# B&R Automation Studio project mappServicesHighlights
Automation Studio 4.9.3.144 SP; mappServices highlights project; technology packages: mapp 5.12.1, mappView 5.12.1, TextSystem 

## Configuration mappDemoDefault

CPU X20CP1301, AutomationRuntime G4.34, Build 4.1.2, Safety 0.0, Vc V4.72.2

### Task classes (Cpu.sw)
```
Cyclic#1:
  Alarm <- Infrastructure.Alarm.prg [disabled]
  WaterHeate <- WaterHeater.prg [disabled]
  Frequenza <- Frequenza.prg
  Program <- Program.prg
Cyclic#2:
  MainContro <- MainControl.prg [disabled]
  PackML <- Industry.PackML.prg [disabled]
  ConveyorSi <- ConveyorSim.prg [disabled]
Cyclic#6:
  Conteggio <- Conteggio.prg
Cyclic#8:
  Sequence <- Infrastructure.Sequence.prg [disabled]
  IO <- Infrastructure.IO.prg [disabled]
  Report <- Infrastructure.Report.prg
  File <- Infrastructure.File.prg [disabled]  // MpFile sample
  Audit <- Infrastructure.Audit.prg [disabled]  // MpAudit Trail sample
  UserH <- Infrastructure.UserH.prg [disabled]  // MpUser sample
  Recipe <- Infrastructure.Recipe.prg  // MRecipe sample
  Energy <- Infrastructure.Energy.prg [disabled]
  CodeBox <- Infrastructure.CodeBox.prg [disabled]
DataObjects: Arnc0sys
Binaries: TCData, udbdef, arsvcreg, mvLoader, TCLang, arflatprv, arcoal, CfgSeq, OpcUaMap, ashwac, sysconf, CfgEnergy, CfgPackML, CfgHistory, Role, User, CfgRecipe, CfgFile, ashwd, CfgAlarm, iomap, CfgAudit, arconfig, TC, CfgUserXLo, CfgWebXs, asfw, CfgUserX, CfgIO, CfgReportF, CfgReport, CfgCodeCor, CfgComUnit, CfgCodeBox, Config, vcgclass, CfgData, CfgOee, CfgSequenc, vccddbox, vccbtn, vcpdvnc, arialbd, vcmgr, vctcal, vcfile, vcctext, vccnum, Visu02, vcfntttf, vcpkat, vcbclass, vccstr, vclibvc, visvc, vccscale, arial, vccshape, vcalarm, vcpfar00, vcclbox, vcdsloc, vcchtml, Visu01, vccdt, vcchspot, vccbmp, vccpopup, Visu03, vcshared, vcxml, vccurl, vcrt, vccslider, vccgauge, vcctrend, vcnet, vccbar, vccpiech, vcdsint, vcpdsw, vccovl, vccline
Libraries: Runtime, Operator, AsIecCon, astime, AsArSdm, DataObj, FileIO, AsBrStr, AsArLog, sys_lib, brsystem, AsArProf, AsMem, AsWStr, standard, AsBrWStr, ArTextSys, MTTypes, MTBasics, MpAlarmX, MpAudit, MpCom, MpEnergy, MpFile, MpIO, MpPackML, MpRecipe, MpReport, MpSequence, MpUserX, MpWebXs, MpCodeBox, MpServer, MpBase, asstring, aruser, asiomman, ashw, asusb, aseth, arssl, arcert, vcresman, areventlog, arproject, powerlnk
```

### Hardware
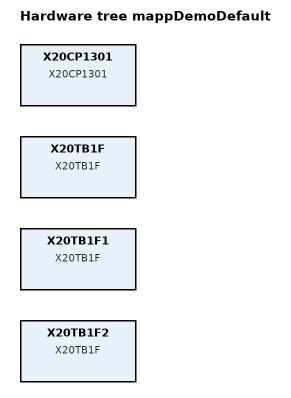
```
X20CP1301 : X20CP1301 v1.7.0.0  [X1 -> X1.SL; X2 -> X2.SL; X3 -> X3.SL]
  Module X1 (Type=X1, Virtual=true, Version=1.7.0.0)
    Connection (Connector=SS1, TargetModule=X20TB1F, TargetConnector=SS)
    Connection (Connector=SL, TargetModule=X20CP1301, TargetConnector=X1)
  Module X2 (Type=X2, Virtual=true, Version=1.7.0.0)
    Connection (Connector=SS1, TargetModule=X20TB1F1, TargetConnector=SS)
    Connection (Connector=SL, TargetModule=X20CP1301, TargetConnector=X2)
  Module X3 (Type=X3, Virtual=true, Version=1.7.0.0)
    Connection (Connector=SS1, TargetModule=X20TB1F2, TargetConnector=SS)
    Connection (Connector=SL, TargetModule=X20CP1301, TargetConnector=X3)
  Connector IF1:
    ActivateIna = 0
  Connector IF2:
    ActivateDevice = 1
    Mode = Manual
    InternetAddress = 192.168.1.38
    SubnetMask = 255.255.255.0
    InaNodeNumber = 0
    Vnc1
    VncKeyMappingFile1 = VC\PS2-Keyboard.dis
    VncMaxConnections1 = 2
    VncRefreshRate1 = 200
  ConfigurationID = mappDemo_CI_Master
  UserPartitionSize = 20
  AutomaticTransferOfUserfiles = on
  RemanentGlobalPvSize = 8192
  VolatileGlobalPvSize = 500000
  CyclicObjects = 300
  BRObjects = 500
  FileDevice1
  FileDeviceName1 = HD
  FileDevicePath1 = C:\
  FileDevice2
  FileDeviceName2 = mappDir
  FileDevicePath2 = C:\mappDemo\CSV
  FileDevice3
  FileDeviceName3 = mappReport
  FileDevicePath3 = C:\mappDemo\Reports\
  FileDevice4
  FileDeviceName4 = mappIO
  FileDevicePath4 = C:\mappDemo\UserFiles\IO
  FileDevice5
  FileDeviceName5 = mappIOBackup
  FileDevicePath5 = C:\mappDemo\UserFiles\IO\Backup
  FileDevice6
  FileDeviceName6 = mappSequence
  FileDevicePath6 = C:\mappDemo\UserFiles\Sequence
  FileDevice7
  FileDeviceName7 = mappCodeBox
  FileDevicePath7 = C:\mappDemo\UserFiles\CodeBox
  FtpUser1
  FtpUsername1 = Promass
  FtpUserPassword1 = NpCmz0K6m8wsjK3Ky3NpfFf+z2PPu3ZJ9pj0GQJGS0g=
  FtpUserSalt1 = EihsEguH
  FTPAccessRight1 = 0
  FTPdevice1 = ALL
  ActivateOpcUa = 1
  OpcUaInformationModels_PV_Version = 1
X20TB1F : X20TB1F v1.0.0.0
X20TB1F1 : X20TB1F v1.0.0.0
X20TB1F2 : X20TB1F v1.0.0.0
```

### IoMap.iom - X20CP1301/IoMap.iom
```iecst
(********************************************************************
 * COPYRIGHT -- Bernecker + Rainer
 ********************************************************************
 * File: IoMap.iom
 * Author: krammerm
 * Created: September 25, 2013
 ********************************************************************
 * IO mapping file
 ********************************************************************)
VAR_CONFIG
	::contatore.Inp_S_Stellare AT %IX."X2".DigitalInput01;
END_VAR
```

### CfgAlarm.mpalarmxcore - X20CP1301/mappServices/CfgAlarm.mpalarmxcore
```
Element gAlarmXCore (Type=mpalarmxcore)
  mapp.AlarmX.Core.Configuration:
    [0]:
      Name = RecordingStarted
      Message = {$mappDemo/MpDataUserAlarm}
      Code = 2501
      Behavior = UserDefined
        AutoReset = TRUE
        Acknowledge = 0
        Recording:
          ActiveToInactive = FALSE
    [1]:
      Name = WaterEmpty
      Message = {$IAT/AlarmWater}
      Code = 2503
      Behavior = LevelMonitoring
        Monitoring:
          MonitoredPV = ::MainContro:Refill.Water
          LowLimitEnable = Static
            Limit = 1
      AdditionalInformation1 = WaterEmpty
    [2]:
      Name = CoffeeEmpty
      Message = {$IAT/AlarmCoffee}
      Code = 2504
      Behavior = LevelMonitoring
        Monitoring:
          MonitoredPV = ::MainContro:Refill.Coffee
          LowLimitEnable = Static
            Limit = 1
      AdditionalInformation1 = CoffeeEmpty
    [3]:
      Name = MilkEmpty
      Message = {$IAT/AlarmMilk}
      Code = 2505
      Behavior = LevelMonitoring
        Monitoring:
          MonitoredPV = ::MainContro:Refill.Milk
          LowLimitEnable = Static
            Limit = 1
      AdditionalInformation1 = MilkEmpty
    [4]:
      Name = SugarEmpty
      Message = {$IAT/AlarmSugar}
      Code = 2506
      Behavior = LevelMonitoring
        Monitoring:
          MonitoredPV = ::MainContro:Refill.Sugar
          LowLimitEnable = Static
            Limit = 1
      AdditionalInformation1 = SugarEmpty
  mapp.AlarmX.Core.Snippets:
    [0]:
      Key = CurrentTemp
      Value:
        PV = ::WaterHeate:WaterHeaterUIConnect.actTemperature
```

### CfgAudit.mpaudittrail - X20CP1301/mappServices/CfgAudit.mpaudittrail
```
Element gAuditTrail (Type=mpaudittrail)
  Audit:
    Events:
      [0] = 16
      [1] = 2
      [2] = 18
      [3] = 17
      [4] = 33
      [5] = 48
      [6] = 64
      [7] = 65
    TextSource = TXT
      OutputFormat = AuditText/Root
      Display = Ne
        Format = AuditDisplayText/DisplayRoot
    Archive = On
    Export:
      FileType = 2
      Encrypt = FALSE
  Alarms = MpAlarmX
```

### CfgCodeBox.mpcodebox - X20CP1301/mappServices/CfgCodeBox.mpcodebox
```
Element CodeBoxCfg (Type=mpcodebox)
  gen:
    progLoc = mappCodeBox
  pvselect:
    0 = 1
      acc = 1
  macro:
    act:
      0:
        id = LampRed
        cd:
          0 = $CodeBox:Lamp.Red := #IN;
      1:
        id = LampYellow
        cd:
          0 = $CodeBox:Lamp.Yellow := #IN;
      2:
        id = LampGreen
        cd:
          0 = $CodeBox:Lamp.Green := #IN;
    cond:
      0:
        id = StartPos
        cd:
          0 = #R := $CodeBox:Cup.StartPosition$;
      1:
        id = CoffeePos
        cd:
          0 = #R := $CodeBox:Cup.CoffeePosition$;
      2:
        id = EndPos
        cd:
          0 = #R := $CodeBox:Cup.EndPosition$;
```

### CfgCodeCor.mpcodeboxcore - X20CP1301/mappServices/CfgCodeCor.mpcodeboxcore
```
Element gCodeBoxCore (Type=mpcodeboxcore)
```

### CfgComUnit.mpcomunit - X20CP1301/mappServices/CfgComUnit.mpcomunit
```
Element gGroup (Type=mpcomunit)
  Display:
    Datapoints:
      0:
        Id = ::Recipe:CoffeeIngredients.Milk
        DisplayUnits:
          Metric:
            Code = MLT
          Imperial:
            Code = MLT
          ImperialUS:
            Code = MLT
      1:
        Id = ::Recipe:CoffeeIngredients.Water
        DisplayUnits:
          Metric:
            Code = MLT
          Imperial:
            Code = MLT
          ImperialUS:
            Code = MLT
      2:
        Id = ::Recipe:CoffeeIngredients.Sugar
        DisplayUnits:
          Metric:
            Code = GRM
          Imperial:
            Code = ONZ
          ImperialUS:
            Code = ONZ
      3:
        Id = ::Recipe:CoffeeIngredients.Coffee
        DisplayUnits:
          Metric:
            Code = GRM
          Imperial:
            Code = ONZ
          ImperialUS:
            Code = ONZ
      4:
        Id = ::Recipe:_Coffee
        DisplayUnits:
          Metric:
            Code = GRM
          Imperial:
            Code = ONZ
          ImperialUS:
            Code = ONZ
      5:
        Id = ::Recipe:_Milk
        DisplayUnits:
          Metric:
            Code = MLT
          Imperial:
            Code = MLT
          ImperialUS:
            Code = MLT
      6:
        Id = ::Recipe:_Sugar
        DisplayUnits:
          Metric:
            Code = GRM
          Imperial:
            Code = ONZ
          ImperialUS:
            Code = ONZ
      7:
        Id = ::Recipe:_Water
        DisplayUnits:
          Metric:
            Code = MLT
          Imperial:
            Code = MLT
          ImperialUS:
            Code = MLT
```

### CfgEnergy.mpenergycore - X20CP1301/mappServices/CfgEnergy.mpenergycore
```
Element gEnergyCore (Type=mpenergycore)
  mapp.energy.collector:
    RecordMemory = 2
    Export:
      FileType:
        ColumnSeparator = ;
  Alarms = MpAlarmX
```

### CfgFile.mpfilemanagerui - X20CP1301/mappServices/CfgFile.mpfilemanagerui
```
Element gFileManagerUI (Type=mpfilemanagerui)
  Alarms = MpAlarmX
```

### CfgHistory.mpalarmxhistory - X20CP1301/mappServices/CfgHistory.mpalarmxhistory
```
Element gAlarmXHistory (Type=mpalarmxhistory)
  mapp.AlarmX.History:
    Auditing = MpAudit
```

### CfgIO.mpio - X20CP1301/mappServices/CfgIO.mpio
```
Element gIoConfig (Type=mpio)
  Import:
    BackupLoc = mappIOBackup
    TemplateLoc = 
  Alarms = MpAlarmX
```

### CfgPackML.mppackmlcore - X20CP1301/mappServices/CfgPackML.mppackmlcore
```
Element gPackMLCore (Type=mppackmlcore)
  Core:
    StartupActiveMode = 1
    Auditing = MpAudit
  Modes:
    Mode[1]:
      ModeID = 1
      Name = Production
      State[1] = 0
      State[5] = 0
      State[10] = 0
      State[11] = 0
      State[12] = 0
      State[13] = 0
      State[14] = 0
      State[17] = 0
    Mode[2]:
      ModeID = 2
  Alarms = MpAlarmX
```

### CfgRecipe.mprecipexml - X20CP1301/mappServices/CfgRecipe.mprecipexml
```
Element gRecipeXml (Type=mprecipexml)
  mapp.Recipe.Xml:
    Auditing = MpAudit
  Alarms = MpAlarmX
```

### CfgReport.mpreportcore - X20CP1301/mappServices/CfgReport.mpreportcore
```
Element gReport (Type=mpreportcore)
  MpReport:
    Settings:
      ResourceDeviceName = HD
      LanguageDependent:
        [0]:
          Language = de
          Font = 1
        [1]:
          Language = en
          Font = 1
    PageLayouts:
      [0]:
        Name = Default
    Styles:
      Text:
        [0]:
          Name = Default
          Size = 12
        [1]:
          Name = Header
          Style = 1
          Size = 20
          Color = FF9900
        [2]:
          Name = Subheader
          Size = 16
          Color = FF9900
      Table:
        [0]:
          Name = Default
          Padding = 10
      Line:
        [0]:
          Name = Default
          Color = FF9900
      Chart:
        PieChart:
          [0]:
            Name = Default
            BorderWidth = 0
        LineChart:
          [0]
        BarChart:
          [0]
    Tables:
      [0]:
        Name = CoffeeInformation
        TableStyle = Default
        TextStyle = Default
        [0]:
          [0] = TextId
            Source = Ora Inizio
            Width = 50
          [1] = DateTime
            Source = ProcessVariable
              ProcessVariable = ::Conteggio:DT_1
            Width = 50
        [1]:
          [0] = TextId
            Source = Ora Fine
            Width = 50
          [1] = DateTime
            Source = ProcessVariable
              ProcessVariable = ::Conteggio:DT_2
            Width = 50
        [2]:
          [0] = TextId
            Source = Tempo Attività
            Width = 50
          [1] = ValueId
            Value:
              ProcessVariable = ::Conteggio:tempo_attuale
            Width = 50
        [3]:
          [0] = TextId
            Source = Giri parziali
            Width = 50
          [1] = ValueId
            Value:
              ProcessVariable = ::contatore.giri_parziali
              UnitDisplay = 1
            Width = 50
        [4]:
          [0] = TextId
            Source = Giri Totali
            Width = 50
          [1] = ValueId
            Value:
              ProcessVariable = ::contatore.giri_totali
              UnitDisplay = 1
            Width = 50
    Contents:
      [0]:
        Name = Discription
        [0]:
          Text = {$Report/ReportDescription}
          TextStyle = Default
      [1]:
        Name = Table
        [0] = Table
          Table = CoffeeInformation
          HorizontalAlign = 1
      [2]:
        Name = Underline
        [0] = Line
          LineStyle = Default
      [3]:
        Name = Header
        [0]:
          Text = {$Report/ReportHeader}
          HorizontalAlign = 1
          TextStyle = Header
      [4]:
        Name = EmptyLine
        [0] = EmptyLine
      [5]:
        Name = EnergyChart
        [0] = Chart
          Chart = Energy
          Width = 60
    Reports:
      [0]:
        Name = Dosaggio
        PageLayout = Default
        Header = Header
        [0]:
          [0]:
            Content = Underline
        [1]:
          [0]:
            Content = EmptyLine
        [2]:
          Heading:
            Text = {$Report/ReportDescriptionHeader}
            TextStyle = Subheader
          [0]:
            Content = Discription
        [3]:
          [0]:
            Content = EmptyLine
        [4]:
          Heading:
            Text = {$Report/ReportHeaderTable}
            TextStyle = Subheader
          [0]:
            Content = Table
        [5]:
          [0]:
            Content = EmptyLine
        [6]:
          [0]:
            Content = EmptyLine
        [7]:
          [0]:
            Content = EnergyChart
  Alarms = MpAlarmX
```

### CfgReportF.mpfilemanagerui - X20CP1301/mappServices/CfgReportF.mpfilemanagerui
```
Element gReportFileManagerUI (Type=mpfilemanagerui)
  Alarms = MpAlarmX
```

### CfgSeq.mpsequencecore - X20CP1301/mappServices/CfgSeq.mpsequencecore
```
Element gSequenceCore (Type=mpsequencecore)
  Sequence:
    DeviceName = mappSequence
    Commands:
      Command[0]:
        Name = SequenceStart
        Text = Start
        Hierarchy = Movement
        CommandType = Movement
          PVStruct = ::Sequence:CmdSeq.Start
      Command[1]:
        Name = SequenceEnd
        Text = End
        Hierarchy = Movement
        CommandType = Movement
          PVStruct = ::Sequence:CmdSeq.Stop
      Command[2]:
        Name = MacroEnd
        Text = EndMakro
        Hierarchy = Movement
      Command[3]:
        Name = Wait
        Text = Wait
        Hierarchy = Movement
        CommandType = Movement
          PVStruct = ::Sequence:CmdSeq.Wait
      Command[4]:
        Name = MoveAxisLeft
        Text = AxisLeft
        Hierarchy = Movement
        CommandType = Movement
          PVStruct = ::Sequence:CmdSeq.AxisLeft
      Command[5]:
        Name = MoveAxisRight
        Text = AxisRight
        Hierarchy = Movement
        CommandType = Movement
          PVStruct = ::Sequence:CmdSeq.AxisRight
          ParStruct = 
      Command[6]:
        Name = Coffee
        Text = Coffee
        Hierarchy = MovementCoffee
        CommandType = Movement
          PVStruct = ::Sequence:CmdSeq.Coffee
      Command[7]:
        Name = TakeOut
        Text = TakeOut
        Hierarchy = MovementCoffee
        CommandType = Movement
          PVStruct = ::Sequence:CmdSeq.TakeOutCup
  Alarms = MpAlarmX
```

### CfgUserX.mpuserx - X20CP1301/mappServices/CfgUserX.mpuserx
```
Element UserMgmtX (Type=mpuserx)
  Groups:
    DefGroup#1:
      id = Administrators
      level = 100
      admin = TRUE
      rights:
        [0] = ViewOnly
        [1] = StartOnly
    DefGroup#2:
      id = Everyone
      level = 1
  Users:
    DefUser#1:
      id = admin
      name = Admin
      lang = en
    DefUser#2:
      id = Anonymous
```

### CfgUserXLo.mpuserxlogin - X20CP1301/mappServices/CfgUserXLo.mpuserxlogin
```
Element gUserXLogin (Type=mpuserxlogin)
  Alarms = MpAlarmX
```

## Logical view

Binary libraries used (declarations not repeated): Runtime, Operator, AsIecCon, AsTime, AsArSdm, DataObj, FileIO, AsBrStr, AsArLog, sys_lib, brsystem, AsWStr, AsArProf, AsMem, standard, AsBrWStr, ArTextSys, MpServer 5.12.0, MpAlarmX 5.12.1, MpBase, MpCodeBox 5.12.1, MpEnergy 5.12.1, MpPackML 5.12.1, MpUserX 5.12.1, MpFile 5.12.1, MpAudit 5.12.1, MpSequence 5.12.1, MpCom, MpIO 5.12.1, MpRecipe 5.12.1, MpWebXs 5.12.1, MpReport 5.12.1, MTBasics, MTTypes, asstring

### Global.typ - Global data types
```iecst
TYPE
	typ_ricetta : 	STRUCT
		Ora_Inizio : DT;
		Ora_Fine : DT;
		Tempo_Attivita : UDINT;
		Giri_Parziali : UDINT;
		Giri_Totali : UDINT;
	END_STRUCT;
	typ_cont : 	STRUCT
		Inp_S_Stellare : BOOL;
		S_stellare : BOOL;
		giri_parziali : UDINT;
		giri_totali : UDINT;
		giri_instant : UDINT;
		frequenza : UDINT;
		nome_ricetta1 : UDINT;
		nome_ricetta2 : STRING[80];
		nome_ricetta3 : UDINT;
		nome_ricetta : STRING[80];
	END_STRUCT;
	PackMLModes :
		(
		PACKML_MODE_PRODUCTION := 1,
		PACKML_MODE_MAINTENANCE := 2
		);
	ReportCoffeeType : 	STRUCT
		Name : STRING[255];
		Water : INT;
		Sugar : INT;
		Coffee : INT;
		Milk : INT;
	END_STRUCT;
	RefillAlarmType : 	STRUCT
		Water : BOOL;
		Sugar : BOOL;
		Milk : BOOL;
		Coffee : BOOL;
	END_STRUCT;
	RefillType : 	STRUCT
		Water : INT;
		Sugar : INT;
		Milk : INT;
		Coffee : INT;
	END_STRUCT;
	CoffeeMainLogicType : 	STRUCT  (*Main logic structure *)
		AxisCupFeeder : CoffeeAxisLogicType; (*Control structure for axis*)
		AxisTakeout : CoffeeAxisLogicType; (*Control structure for axis*)
		cmdAbort : BOOL; (*HMI control to start the brewing process*)
		cmdStop : BOOL; (*HMI control to start the brewing process*)
		cmdClear : BOOL; (*HMI control to start the brewing process*)
		cmdStart : BOOL; (*HMI control to start the brewing process*)
		TemperatureWithinLimit : BOOL; (*HMI control bit *)
		CreateFirstRecipe : BOOL; (*Enable synchronization when creating the default recipes*)
		visPictureIndex : USINT; (*RecipeIndex when creating the default recipes*)
		cmdTakeout : BOOL;
		Refill : RefillType; (*Structure to control the ingredients*)
		AlarmRefill : RefillAlarmType; (*Structure which is controlling the Refill-Alarms*)
		CoffeeState : CoffeeStateEnum;
		ReportCoffee : ARRAY[0..199]OF ReportCoffeeType;
		PackMLState : STRING[80];
		IdleState : BOOL;
	END_STRUCT;
	CoffeeAxisLogicType : 	STRUCT  (*Sub structure for controlling axis*)
		Active : BOOL; (*Axis component is ready*)
		Power : BOOL; (*Power on command*)
		PowerOn : BOOL; (*Power is on*)
		Home : BOOL; (*Homing command *)
		MoveAdditive : BOOL; (*MoveAdditive command*)
		MoveActive : BOOL; (*Move active*)
		InPosition : BOOL; (*Commanded position reached *)
		Position : LREAL; (*Current position*)
	END_STRUCT;
	CoffeeStateEnum :
		(
		COFFEE_WAIT := 0,
		COFFEE_TAKEWATER := 1,
		COFFEE_TAKECOFFEE := 2,
		COFFEE_TAKECOFFEEMILK := 3,
		COFFEE_RELEASE := 4,
		COFFEE_FINISH := 5
		);
END_TYPE
```

### Global.var - Global variables
```iecst
(*Definitions for main components of the coffee machine*)
VAR
	Ricetta : typ_ricetta := (0);
	MpReportCore_0 : MpReportCore := (0); (*Core variable for MpReport*)
	t_ok : BOOL := FALSE;
	CTU_1 : CTU := (0);
	StartGenerate : BOOL := 0; (*variable for interaction with Visualization*)
	gClearAlarm : BOOL := FALSE; (*Check if Alarm can be cleared*)
	gCoffeeMainLogic : CoffeeMainLogicType; (*Control structure of main logic*)
	gSetLanguage : STRING[80] := ''; (*Set the current language*)
	contatore : typ_cont := (0);
END_VAR
```


### Package Logical/Infrastructure - Infrastructure Components

### Program Logical/Infrastructure/Alarm (IEC) - Alarm handling

#### Main.st
```iecst
PROGRAM _CYCLIC

	//Set FB parameter:
	MpAlarmXCore_0(
		Enable := TRUE,
		MpLink := ADR(gAlarmXCore));

	MpAlarmXListUI_0(
		MpLink := ADR(gAlarmXCore),
		Enable := TRUE,
		UIConnect := ADR(MpAlarmXListUIConnect));

	MpAlarmXHistory_0(
		MpLink := ADR(gAlarmXHistory),
		Enable := TRUE,
		DeviceName := ADR('mappDir'),
		Language := ADR(gSetLanguage));

	//Show Alarm-Button in Visualization
	IF MpAlarmXCore_0.ActiveAlarms <> 0 OR MpAlarmXCore_0.PendingAlarms <> 0 THEN
		AlarmButton := 1;
		gCoffeeMainLogic.cmdAbort := TRUE;
		gCoffeeMainLogic.cmdClear := FALSE;
	ELSE
		AlarmButton := 0;
		gCoffeeMainLogic.cmdClear := TRUE;
		gCoffeeMainLogic.cmdAbort := FALSE;
	END_IF

	IF gCoffeeMainLogic.IdleState AND AlarmButton = 0 THEN
		ChangeStyleAlarmButton := 1;
	ELSE
		ChangeStyleAlarmButton := 0;
	END_IF

	IF MpAlarmXHistory_0.CommandDone = TRUE THEN
		MpAlarmXHistory_0.Export := FALSE;
	END_IF

	//Set Alarm-Video
	IF brsstrcmp(ADR(AlarmVideo), ADR("")) = 0 THEN
		AlarmInfo := FALSE;
	ELSE
		AlarmInfo := TRUE;
	END_IF

	FilterConfiguration;
	SortConfiguration;
	HistoryFilter;
	HistorySort;

END_PROGRAM

PROGRAM _EXIT

	//Disable FBs
	MpAlarmXCore_0(Enable := FALSE);
	MpAlarmXHistory_0(Enable := FALSE);
	MpAlarmXHistoryUI_0(Enable := FALSE);
	MpAlarmXListUI_0(Enable := FALSE);

END_PROGRAM
```

#### Variables.var - Local variables
```iecst
VAR
	MpAlarmXHistory_0 : MpAlarmXHistory; (*MpAlarmXHistory instance*)
	MpAlarmXHistoryUI_0 : MpAlarmXHistoryUI; (*MpAlarmXHistoryUI instance*)
	MpAlarmXListUI_0 : MpAlarmXListUI; (*MpAlarmXList instance*)
	MpAlarmXCore_0 : MpAlarmXCore; (*MpAlarmXCore instance*)
	ChangeStyleAlarmButton : USINT := 0; (*changeStyle of a AlarmFlyout in mappView*)
	AlarmButton : BOOL := FALSE; (*Contol Variable for Button in mapp View*)
	MpAlarmXListUIConnect : MpAlarmXListUIConnectType := (0);
	AlarmVideo : WSTRING[255] := "";
	AlarmInfo : BOOL := 0;
	FilterConfiguration : STRING[1000] := '';
	SortConfiguration : STRING[1000] := '';
	HistoryFilter : STRING[2000] := '';
	HistorySort : STRING[2000] := '';
END_VAR
```

### Program Logical/Infrastructure/Recipe (IEC) - Recipe handling

#### Cyclic.ld - Cyclic code
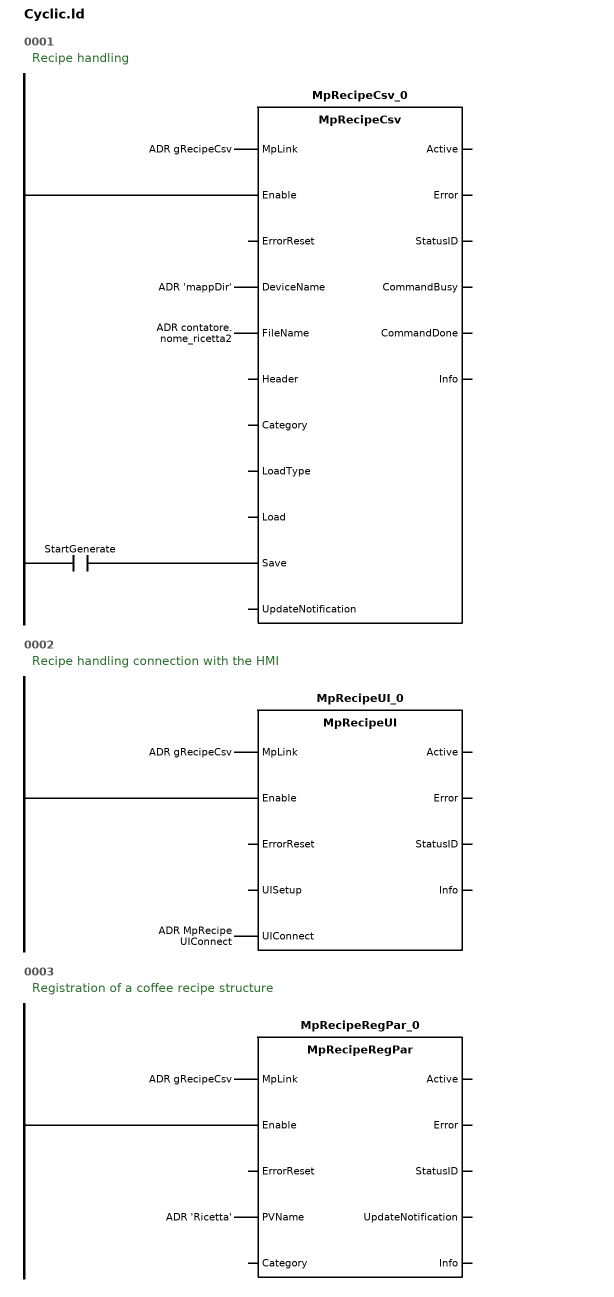
Ladder, written as Structured Text:
```iecst
PROGRAM _CYCLIC
(* Network 1: Recipe handling *)
MpRecipeCsv_0(MpLink := ADR(gRecipeCsv), Enable := TRUE, DeviceName := ADR('mappDir'), FileName := ADR(contatore.nome_ricetta2), Save := StartGenerate);

(* Network 2: Recipe handling connection with the HMI *)
MpRecipeUI_0(MpLink := ADR(gRecipeCsv), Enable := TRUE, UIConnect := ADR(MpRecipeUIConnect));

(* Network 3: Registration of a coffee recipe structure *)
MpRecipeRegPar_0(MpLink := ADR(gRecipeCsv), Enable := TRUE, PVName := ADR('Ricetta'));
END_PROGRAM
```

#### Init.ld - Init code
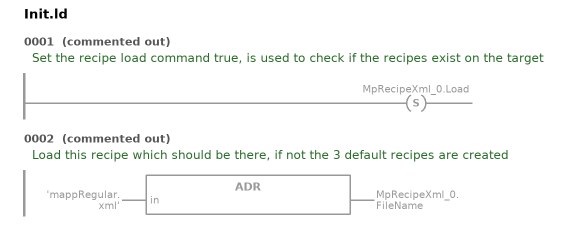
Ladder, written as Structured Text:
```iecst
PROGRAM _INIT
(* Network 1: Set the recipe load command true, is used to check if the recipes exist on the target *) (* commented out *)
// MpRecipeXml_0.Load := TRUE;

(* Network 2: Load this recipe which should be there, if not the 3 default recipes are created *) (* commented out *)
// MpRecipeXml_0.FileName := ADR(in := 'mappRegular.xml');
END_PROGRAM
```

#### Exit.ld
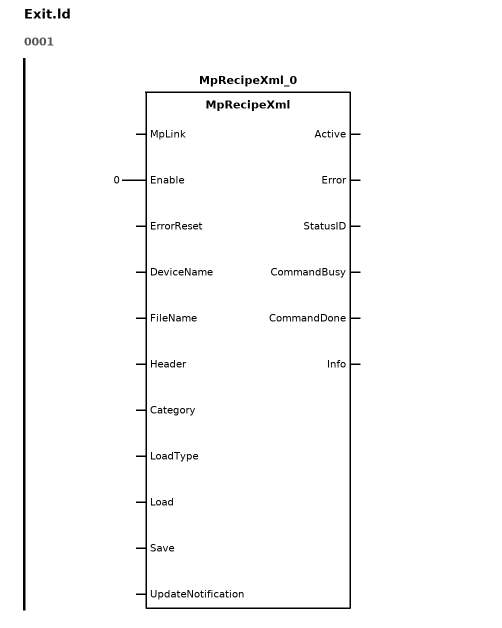
Ladder, written as Structured Text:
```iecst
PROGRAM _EXIT
(* Network 1 *)
MpRecipeXml_0(Enable := 0);
END_PROGRAM
```

#### Variables.var - Local variables
```iecst
VAR
	MpRecipeRegPar_0 : MpRecipeRegPar; (*Registration of the recipe structure variable*)
	MpRecipeUI_0 : MpRecipeUI := (UISetup:=(RecipeListSize:=12,Confirmation:=(RecipeLoad:=0,RecipeSave:=0,RecipeCreate:=0,RecipeDelete:=TRUE))); (*MpRecipeUI Component*)
	MpRecipeCsv_0 : MpRecipeCsv := (0);
	MpRecipeXml_0 : MpRecipeXml; (*Recipe Handling FUB*)
	RecipeCreateStep : RecipeCreateSteps := IDLE; (*Internal variable for recipe creating state machine*)
	MpRecipeUIConnect : MpRecipeUIConnectType := (Recipe:=(Filter:='*xml'),New:=(FileName:='newRecipe.xml')); (*MpRecipeUI connection datapoints*)
	CoffeeIngredients : CoffeeIngredientsType := (Milk:=100,Water:=150,Sugar:=30,Coffee:=60); (*Coffee machine recipe structure*)
END_VAR
(*Variables for AuditTrail*)
VAR
	MpAuditValueChangeStatus : DINT; (*Status variable for MpAuditValueChange function*)
	_Water : INT := 0;
	_Sugar : INT := 0;
	_Milk : INT := 0;
	_Coffee : INT := 0;
	_SelectedIndex : UINT := 800;
END_VAR
```

#### Types.typ - Local Variables
```iecst
TYPE
	RecipeCreateSteps :
		( (*Steps for creating recipes*)
		IDLE := 0, (*Idle State *)
		CREATE_1 := 10, (*Create coffee mappRegular*)
		DONE_1 := 11, (*mappRegular was created*)
		CREATE_2 := 20, (*Create coffee mappEspresso*)
		DONE_2 := 21, (*mappEspresso was created*)
		CREATE_3 := 30, (*Create coffee mappCappuccino*)
		DONE_3 := 31, (*mappCappuccino was created*)
		CREATE_4 := 40, (*Create coffee mappMilkCoffee*)
		DONE_4 := 41, (*mappMilkCoffee was created*)
		ALL_DONE := 50 (*All recipes were created*)
		);
	CoffeeIngredientsType : 	STRUCT  (*Main ingredients structure*)
		Milk : INT; (*Amount of milk per cup*)
		Water : INT; (*Amount of water per cup*)
		Sugar : INT; (*Amount of sugar per cup*)
		Coffee : INT; (*Amount of coffee per cup*)
	END_STRUCT;
END_TYPE
```

#### CreateRecipes.st - Create recipes for the first time the project runs
```iecst
ACTION CreateRecipes:

	// create default recipes in case they don't exist yet on the target
	// recipes are created by using the the MpRecipeXml instance interface

	CASE RecipeCreateStep OF
		IDLE:	// check for load error > triggers the default creation > if no error everything is ready to go
			IF (MpRecipeUIConnect.Recipe.List.Names[0] = '') THEN
				MpRecipeXml_0.Load 			:= FALSE;
				MpRecipeXml_0.ErrorReset 	:= TRUE;
				RecipeCreateStep 			:= CREATE_1;
			ELSE
				MpRecipeUIConnect.Recipe.Load := TRUE;
			END_IF

			// reset the load command from the init when recipe was loaded successfully
			IF (MpRecipeXml_0.CommandDone) AND (MpRecipeXml_0.Load = TRUE) THEN
				MpRecipeXml_0.Load 				:= FALSE;
			END_IF

		CREATE_1:	// create the first recipe with default values, file name and a known picture index (Bitmap Group in the HMI)
			MpRecipeXml_0.ErrorReset 			:= FALSE;

			gCoffeeMainLogic.CreateFirstRecipe 	:= TRUE;
			gCoffeeMainLogic.visPictureIndex	:= 1;
			CoffeeIngredients.Milk 				:= 0;
			CoffeeIngredients.Water 			:= 150;
			CoffeeIngredients.Sugar 			:= 0;
			CoffeeIngredients.Coffee 			:= 60;
			MpRecipeXml_0.FileName 				:= ADR('mappRegular.xml');
			MpRecipeXml_0.Save					:= TRUE;
			RecipeCreateStep 					:= DONE_1;

		DONE_1:	// when CommandDone GoTo next step
			IF(MpRecipeXml_0.CommandDone) THEN
				RecipeCreateStep 			:= CREATE_2;
				MpRecipeXml_0.Save			:= FALSE;
			END_IF;

		CREATE_2:	// create the next recipe with default values, file name and a known picture index (Bitmap Group in the HMI)

			gCoffeeMainLogic.visPictureIndex	:= 2;
			CoffeeIngredients.Milk 				:= 0;
			CoffeeIngredients.Water 			:= 75;
			CoffeeIngredients.Sugar 			:= 0;
			CoffeeIngredients.Coffee 			:= 120;
			MpRecipeXml_0.FileName 				:= ADR('mappEspresso.xml');
			MpRecipeXml_0.Save					:= TRUE;
			RecipeCreateStep 					:= DONE_2;

		DONE_2:	// when CommandDone GoTo next step
			IF (MpRecipeXml_0.CommandDone) THEN
				RecipeCreateStep 			:= CREATE_3;
				MpRecipeXml_0.Save			:= FALSE;
			END_IF;

		CREATE_3:	// create the next recipe with default values, file name and a known picture index (Bitmap Group in the HMI)

			gCoffeeMainLogic.visPictureIndex	:= 3;
			CoffeeIngredients.Milk 				:= 75;
			CoffeeIngredients.Water 			:= 75;
			CoffeeIngredients.Sugar 			:= 20;
			CoffeeIngredients.Coffee 			:= 120;
			MpRecipeXml_0.FileName 				:= ADR('mappCappuccino.xml');
			MpRecipeXml_0.Save					:= TRUE;
			RecipeCreateStep 					:= DONE_3;

		DONE_3:	// when CommandDone creating recipes is done
			IF(MpRecipeXml_0.CommandDone) THEN
				RecipeCreateStep 					:= CREATE_4;
				MpRecipeXml_0.Save					:= FALSE;
			END_IF;
		CREATE_4:	// create the next recipe with default values, file name and a known picture index (Bitmap Group in the HMI)

			gCoffeeMainLogic.visPictureIndex	:= 3;
			CoffeeIngredients.Milk 				:= 100;
			CoffeeIngredients.Water 			:= 50;
			CoffeeIngredients.Sugar 			:= 0;
			CoffeeIngredients.Coffee 			:= 60;
			MpRecipeXml_0.FileName 				:= ADR('mappMilkCoffee.xml');
			MpRecipeXml_0.Save					:= TRUE;
			MpRecipeUIConnect.Recipe.Refresh 	:= TRUE;
			RecipeCreateStep 					:= DONE_4;

		DONE_4:	// when CommandDone creating recipes is done
			IF(MpRecipeXml_0.CommandDone) THEN
				RecipeCreateStep 					:= ALL_DONE;
				MpRecipeXml_0.Save					:= FALSE;
				gCoffeeMainLogic.CreateFirstRecipe 	:= FALSE;
				MpRecipeUIConnect.Recipe.Refresh 	:= FALSE;
			END_IF;
	END_CASE;

END_ACTION
```

#### AuditTrail.st - Watch recipe variable for value change
```iecst
ACTION AuditTrail:

	// Watch for changes in coffee
	IF (CoffeeIngredients.Coffee <> _Coffee) THEN
		MpAuditValueChangeStatus := MpAuditValueChange(gAuditTrail, _Coffee, CoffeeIngredients.Coffee, '100');
		_Coffee 				 := CoffeeIngredients.Coffee;
	END_IF

	// Watch for changes in milk
	IF (CoffeeIngredients.Milk <> _Milk) THEN
		MpAuditValueChangeStatus := MpAuditValueChange(gAuditTrail, _Milk, CoffeeIngredients.Milk, '101');
		_Milk 					 := CoffeeIngredients.Milk;
	END_IF

	// Watch for changes in sugar
	IF (CoffeeIngredients.Sugar <> _Sugar) THEN
		MpAuditValueChangeStatus := MpAuditValueChange(gAuditTrail, _Sugar, CoffeeIngredients.Sugar, '102');
		_Sugar 					 := CoffeeIngredients.Sugar;
	END_IF

	// Watch for changes in water
	IF (CoffeeIngredients.Water <> _Water) THEN
		MpAuditValueChangeStatus := MpAuditValueChange(gAuditTrail, _Water, CoffeeIngredients.Water, '103');
		_Water 					 := CoffeeIngredients.Water;
	END_IF

	//Load new recipe set recipe parameters
	IF MpRecipeUIConnect.Recipe.List.SelectedIndex <> _SelectedIndex THEN
		_SelectedIndex := MpRecipeUIConnect.Recipe.List.SelectedIndex;
		MpRecipeUIConnect.Recipe.Load := TRUE;

	END_IF

	gCoffeeMainLogic.Refill.Coffee := CoffeeIngredients.Coffee ;
	gCoffeeMainLogic.Refill.Milk := CoffeeIngredients.Milk ;
	gCoffeeMainLogic.Refill.Sugar := CoffeeIngredients.Sugar ;
	gCoffeeMainLogic.Refill.Water := CoffeeIngredients.Water ;

END_ACTION
```

### Program Logical/Infrastructure/File (IEC) - File manager

#### Cyclic.ld - Cyclic code
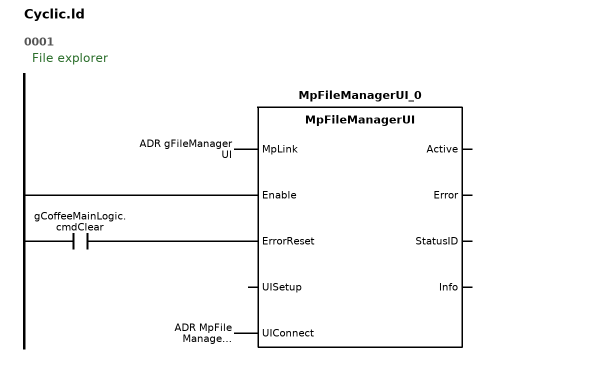
Ladder, written as Structured Text:
```iecst
PROGRAM _CYCLIC
(* Network 1: File explorer *)
MpFileManagerUI_0(MpLink := ADR(gFileManagerUI), Enable := TRUE, ErrorReset := gCoffeeMainLogic.cmdClear, UIConnect := ADR(MpFileManagerUIConnect));
END_PROGRAM
```

#### Init.ld - Init code
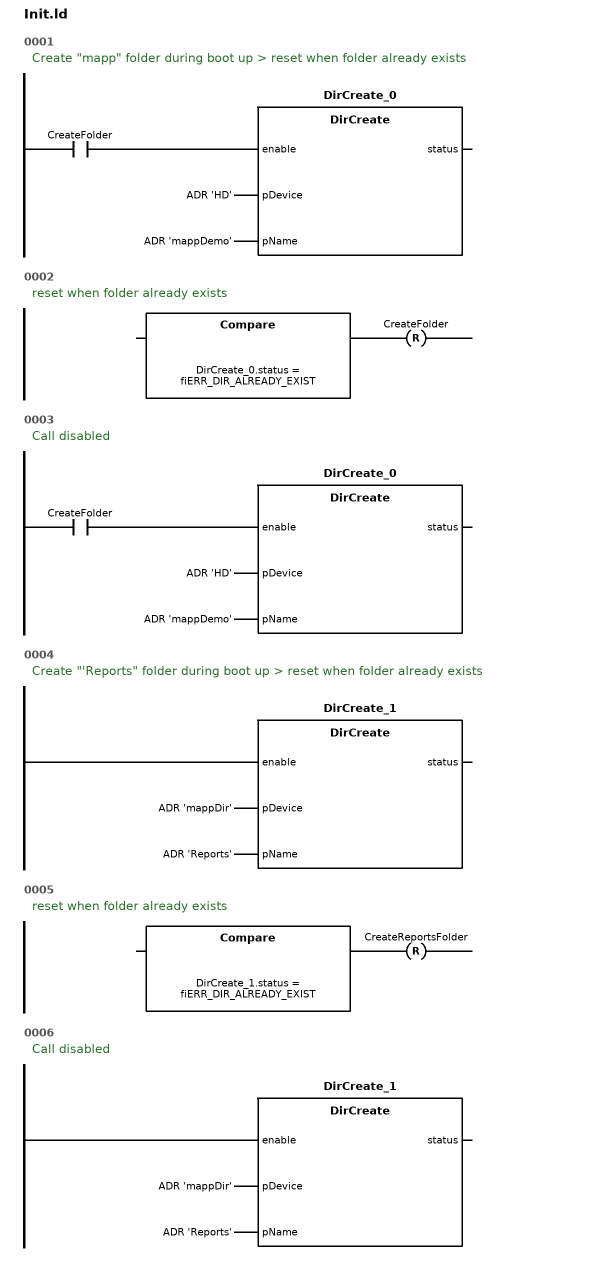
Ladder, written as Structured Text:
```iecst
PROGRAM _INIT
(* Network 1: Create "mapp" folder during boot up > reset when folder already exists  *)
DirCreate_0(enable := CreateFolder, pDevice := ADR('HD'), pName := ADR('mappDemo'));

(* Network 2: reset when folder already exists  *)
IF (DirCreate_0.status = fiERR_DIR_ALREADY_EXIST) THEN CreateFolder := FALSE; END_IF;

(* Network 3: Call disabled *)
DirCreate_0(enable := CreateFolder, pDevice := ADR('HD'), pName := ADR('mappDemo'));

(* Network 4: Create "'Reports" folder during boot up > reset when folder already exists  *)
DirCreate_1(enable := TRUE, pDevice := ADR('mappDir'), pName := ADR('Reports'));

(* Network 5: reset when folder already exists  *)
IF (DirCreate_1.status = fiERR_DIR_ALREADY_EXIST) THEN CreateReportsFolder := FALSE; END_IF;

(* Network 6: Call disabled *)
DirCreate_1(enable := TRUE, pDevice := ADR('mappDir'), pName := ADR('Reports'));
END_PROGRAM
```

#### Variables.var - Local variables
```iecst
VAR
	MpFileManagerUI_0 : MpFileManagerUI; (*MpFileManagerUI instanz*)
	DirCreate_0 : DirCreate; (*FileIO function block for creating the folder "mapp" in case it does not exist yet*)
	CreateFolder : BOOL := TRUE; (*Control bit*)
	MpFileManagerUIConnect : MpFileManagerUIConnectType := (DeviceList:=(DeviceNames:=['mappDir',9('')])); (*MpFileManagerUI connection datapoints*)
	CreateReportsFolder : BOOL := 0;
	DirCreate_1 : DirCreate := (0);
END_VAR
```

### Program Logical/Infrastructure/Audit (IEC) - AuditTrail handling

#### Cyclic.st - Implementation code
```iecst
PROGRAM _CYCLIC

	//Set FB parameters
	MpAuditTrail_0(
		MpLink := ADR(gAuditTrail),
		Enable := TRUE, DeviceName := ADR('mappDir'),
		ErrorReset := gCoffeeMainLogic.cmdClear,
		Language := ADR(gSetLanguage));

	MpAuditTrailUI_0(
		MpLink := ADR(gAuditTrail),
		Enable := TRUE,
		UIConnect := ADR(MpAuditTrailUIConnect),
		ErrorReset := gCoffeeMainLogic.cmdClear,
		Language := ADR(gSetLanguage));

	IF (MpAuditTrail_0.Export) AND (MpAuditTrail_0.CommandDone) THEN
		MpAuditTrail_0.Export := FALSE;
	END_IF

	IF MpAuditTrail_0.ArchiveAvailable THEN
		MpAuditTrail_0.ExportArchive := TRUE;
	ELSE
		MpAuditTrail_0.ExportArchive := FALSE;
	END_IF

	FilterConfiguration;
	SortConfiguraiton;

END_PROGRAM
PROGRAM _EXIT

	//Disable FBs
	MpAuditTrail_0(Enable := FALSE);
	MpAuditTrailUI_0(Enable := FALSE);

END_PROGRAM
```

#### Variables.var - Local variables
```iecst
VAR
	MpAuditTrail_0 : MpAuditTrail; (*Parent component for change tracking*)
	MpAuditTrailUI_0 : MpAuditTrailUI := (UISetup:=(EventListSize:=20)); (*VC4 page connection  *)
	MpAuditTrailUIConnect : MpAuditTrailUIConnectType := (Filter:=(Dialog:=(From:=(Year:=1970,Month:=1,Day:=1,Hour:=00,Minute:=00),Until:=(Year:=1970,Month:=1,Day:=1,Hour:=00,Minute:=00)))); (*MpAuditTrailUI connection datapoints*)
	lng : STRING[80] := '';
	FilterConfiguration : STRING[2000] := '';
	SortConfiguraiton : STRING[2000] := '';
END_VAR
```

### Program Logical/Infrastructure/UserH (IEC) - User handling

#### Main.st
```iecst
PROGRAM _INIT

	LoginAsDefault := FALSE;

END_PROGRAM
PROGRAM _CYCLIC

	//Set FB parameters
	MpUserXLogin_0(
		Enable := TRUE,
		MpLink := ADR(gUserXLogin),
		UserName := ADR(LOGIN_AS_DEFAULT_USERNAME),
		Password := ADR(LOGIN_AS_DEFAULT_PASSWORD));

	MpUserXManagerUI_0(
		Enable := TRUE,
		MpLink := ADR(gUserXLogin),
		UIConnect := ADR(MpUserXManagerUIConnect));

	MpUserXLoginUI_0(
		Enable := TRUE,
		UIConnect := ADR(MpUserXLoginUIConnect),
		MpLink := ADR(gUserXLogin));

	//Call Action
	mappViewConnection;

END_PROGRAM
PROGRAM _EXIT

	//Disable FBs
	MpUserXLogin_0(Enable := FALSE, Login := FALSE);
	MpUserXManagerUI_0(Enable := FALSE);
	MpUserXLoginUI_0(Enable := FALSE);

END_PROGRAM
```

#### mappViewConnection.st - Connection to mapp View
```iecst
ACTION mappViewConnection:

		//Set Login command to FALSE;
	IF MpUserXLogin_0.CommandDone = TRUE THEN
		MpUserXLogin_0.Login := FALSE;
		DeleteTextInput := TRUE ;
	END_IF;

	//Log in as Anonymous
	IF MpUserXLogin_0.CurrentLevel = 0 THEN
		TON_0(IN := TRUE, PT := T#1s5ms);
	ELSIF MpUserXLogin_0.CurrentLevel > 0 THEN
		TON_0(IN := FALSE, PT := T#1s5ms);
	END_IF

	IF ((MpUserXLogin_0.CurrentLevel = 0) AND (LoginAsDefault = TRUE)) OR TON_0.Q = TRUE THEN
		TON_0(IN := FALSE, PT := T#1s5ms);
		MpUserXLogin_0.UserName := ADR(LOGIN_AS_DEFAULT_USERNAME);
		MpUserXLogin_0.Password := ADR(LOGIN_AS_DEFAULT_PASSWORD);
		MpUserXLogin_0.Login := TRUE;
		LoginAsDefault := FALSE;
	END_IF;

	//Set Role in Visualization
	IF MpUserXLogin_0.CurrentLevel = 100 THEN
		Role := 'Administrator';

	ELSIF MpUserXLogin_0.CurrentLevel = 50 THEN
		Role := 'Supervisor';

	ELSIF MpUserXLogin_0.CurrentLevel = 10 THEN
		Role := 'Operator';
	ELSE
		Role := 'Anonymous';
	END_IF

	// Logout in mappView with valuechange in Eventbinding
	IF MpUserXLoginUIConnect.MessageBox.ErrorNumber = 28672 OR MpUserXLoginUIConnect.MessageBox.ErrorNumber = 28673 OR MpUserXLoginUIConnect.MessageBox.ErrorNumber = 28680 THEN
		MappViewLogout := 1;
	ELSIF MpUserXLoginUIConnect.MessageBox.ErrorNumber = 0 THEN
		MappViewLogout := 0;
	END_IF

	IF MpUserXLoginUIConnect.MessageBox.ErrorNumber <> 0 THEN
		ShowErrorLoginDialog := TRUE;
	ELSE
		ShowErrorLoginDialog := FALSE;
	END_IF

END_ACTION
```

#### Variables.var - Local variables
```iecst
VAR CONSTANT
	LOGIN_AS_DEFAULT_USERNAME : WSTRING[20] := "Anonymous"; (*Constant for auto login*)
	LOGIN_AS_DEFAULT_PASSWORD : WSTRING[20] := ""; (*Constant for auto login*)
END_VAR
VAR
	MpUserXManagerUI_0 : MpUserXManagerUI; (*MpUserXManagerUI FUB*)
	MpUserXManagerUIConnect : {REDUND_UNREPLICABLE} MpUserXMgrUIConnectType; (*MpUserXManagerUI connection datapoints*)
	MpUserXLogin_0 : MpUserXLogin := (0); (*MpUserXLogin FUB*)
	MpUserXLoginUI_0 : MpUserXLoginUI := (0); (*MpUserXLoginUI FUB*)
	MpUserXLoginUIConnect : MpUserXLoginUIConnectType := (0); (*MpUserXLoginUI connection datapoints*)
	LoginAsDefault : BOOL := 0; (*trigger login as Anonymous *)
	TON_0 : TON := (0); (*Timer wait for login else login as default*)
	DeleteTextInput : BOOL := 0;
	Role : STRING[80] := '0';
	MappViewLogout : INT := 0;
	ShowErrorLoginDialog : BOOL := 0;
END_VAR
```

### Program Logical/Infrastructure/Energy (IEC) - Energy handling

#### Cyclic.ld - Cyclic code
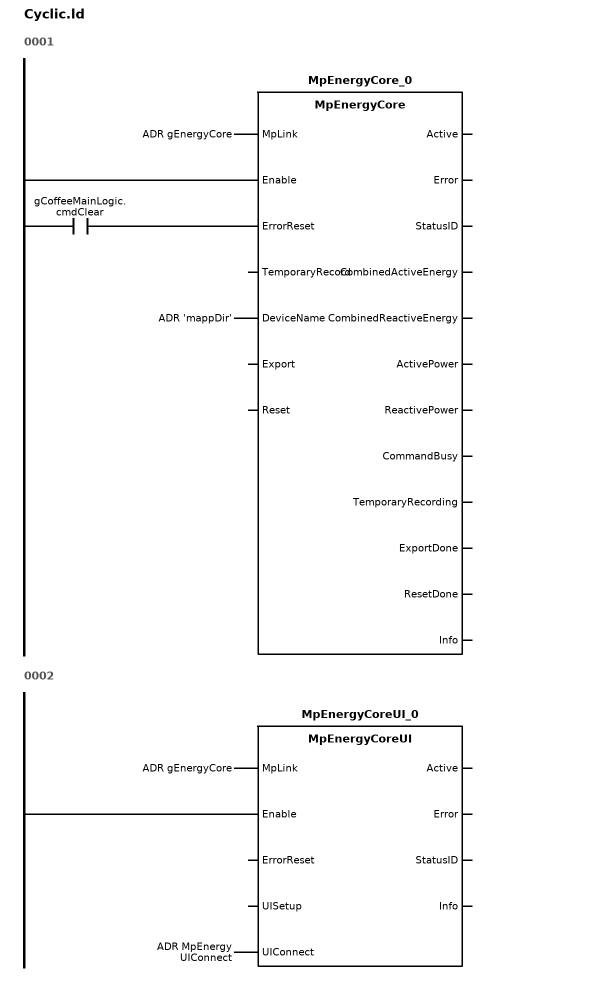
Ladder, written as Structured Text:
```iecst
PROGRAM _CYCLIC
(* Network 1 *)
MpEnergyCore_0(MpLink := ADR(gEnergyCore), Enable := TRUE, ErrorReset := gCoffeeMainLogic.cmdClear, DeviceName := ADR('mappDir'));

(* Network 2 *)
MpEnergyCoreUI_0(MpLink := ADR(gEnergyCore), Enable := TRUE, UIConnect := ADR(MpEnergyUIConnect));
END_PROGRAM
```

#### Exit.ld
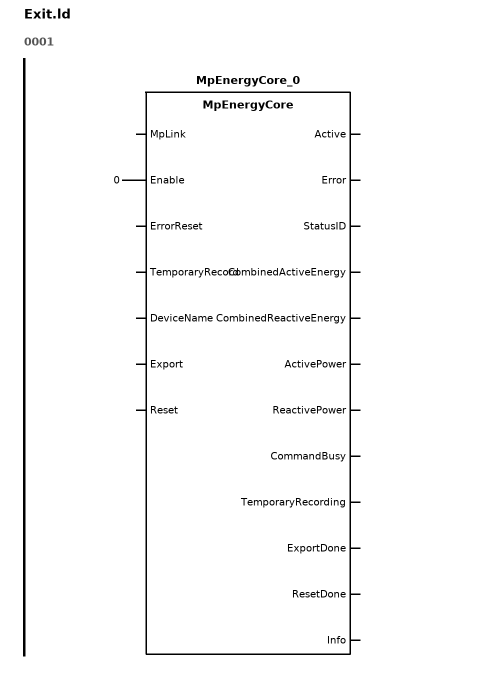
Ladder, written as Structured Text:
```iecst
PROGRAM _EXIT
(* Network 1 *)
MpEnergyCore_0(Enable := 0);
END_PROGRAM
```

#### Variables.var - Local variables
```iecst
VAR
	MpEnergyCore_0 : MpEnergyCore; (*MpEnergyCore instance*)
	MpEnergyCoreUI_0 : MpEnergyCoreUI := (UISetup:=(ModuleListSize:=6)); (*MpEnergyCoreUI instance*)
	MpEnergyUIConnect : MpEnergyCoreUIConnectType; (*MpEnergyUI connection datapoints*)
END_VAR
```

### Program Logical/Infrastructure/Report (IEC) - Report handling

#### Main.st - Cyclic code
```iecst
PROGRAM _CYCLIC

	//Call FBs:
	MpReportCore_0(
		Enable := TRUE,
		MpLink := ADR(gReport),
		Name := ADR(REPORT_NAME),
		DeviceName := ADR(REPORT_DEVICE));
		MpFileManagerUI_0(Enable := TRUE);

	//Call Action
	RefreshReport;

END_PROGRAM
PROGRAM _EXIT

	//Disable FBs
	MpReportCore_0(Enable := FALSE);
	MpFileManagerUI_0(Enable := FALSE);

END_PROGRAM
```

#### Variables.var - Local variables
```iecst
VAR CONSTANT
	STR_FILE_DEVICE : STRING[80] := '/FileDevice:mappReport/';
END_VAR
VAR
	LanguageSelect_0 : LanguageSelect := (LanguageSelection:=['en','de'],SelectedIndex:=0);
	MpFileManagerUI_0 : MpFileManagerUI;
	MpFileManagerUIConnect : MpFileManagerUIConnectType := (DeviceList:=(DeviceNames:=['mappReport',9('')]));
END_VAR
VAR CONSTANT
	REPORT_DEVICE : STRING[80] := 'mappReport'; (*Constant contains filedevice for save reports *)
	REPORT_NAME : STRING[80] := 'Dosaggio'; (*Constant contains name of Report*)
END_VAR
VAR
	DisplayFileName : ARRAY[0..49] OF STRING[255] := [50('')]; (*Displayed Files for mappView*)
	StrSelectedFile : STRING[256] := '0'; (*Gives the path of selected report to pdfViewer in mappView*)
	EnableGenerate : BOOL := TRUE; (*HMI control bit*)
	EnableDelete : BOOL := TRUE; (*HMI control bit*)
	i : USINT := 0; (*index for save filenames in a array*)
	DisplayFileNameIndex : USINT := 0; (*index of selected file for display in table in mappView*)
	DeleteReport : BOOL := 0; (*Start deleting a Report*)
	Refresh : BOOL := 0; (*strrt refresh process*)
	TON_0 : TON := (0); (*Timer to wait before refresh*)
END_VAR
```

#### RefreshReport.st - Showing Report in list
```iecst
ACTION RefreshReport:

	MpFileManagerUI_0.MpLink := ADR(gReportFileManagerUI);
	MpFileManagerUI_0.UIConnect := ADR(MpFileManagerUIConnect);

	IF StartGenerate = TRUE THEN		//Generate process
		MpReportCore_0.Language := ADR(LanguageSelect_0.LanguageSelection[LanguageSelect_0.SelectedIndex]);
		MpReportCore_0.Generate := TRUE;

		IF MpReportCore_0.CommandDone = TRUE THEN

			StartGenerate := FALSE;
			Refresh := TRUE;
			EnableGenerate := FALSE;
		END_IF

	ELSE
		MpReportCore_0.Generate := FALSE;
	END_IF

	IF DeleteReport = TRUE THEN				//Deleting process
		MpFileManagerUIConnect.File.Delete := TRUE;
		MpFileManagerUIConnect.MessageBox.Confirm := TRUE;
		DeleteReport := FALSE;
		Refresh := TRUE;
		EnableDelete := FALSE;
	END_IF

	IF Refresh = TRUE THEN				//Refresh process
		TON_0(IN := TRUE, PT := T#2s);
		IF TON_0.Q = TRUE THEN
			Refresh := FALSE;
			TON_0(IN := FALSE, PT := T#2s);
			MpFileManagerUIConnect.File.Refresh := TRUE;
		END_IF
	END_IF

	IF Refresh = FALSE THEN		//reset enable attribute for buttons
		EnableDelete := TRUE;
		EnableGenerate := TRUE;
	END_IF

	FOR i := 0 TO 49 DO							// Save Filenames to a seperate array for display in Table
		DisplayFileName[i] := MpFileManagerUIConnect.File.List.Items[i].Name;
		IF DisplayFileNameIndex = i THEN		// if selected set a index for display selected file in table
			MpFileManagerUIConnect.File.List.Items[i].IsSelected := TRUE;
		END_IF
	END_FOR

	StrSelectedFile := CONCAT(STR_FILE_DEVICE, MpFileManagerUIConnect.File.List.Items[DisplayFileNameIndex].Name);		// String for pdfViewer to display right report

	IF LanguageSelect_0.SelectedIndex = 0 THEN
		gSetLanguage := 'en';
	ELSE
		gSetLanguage := 'de';
	END_IF

END_ACTION
```

### Program Logical/Infrastructure/IO (IEC) - Hardware handling

#### Main.st - Cyclic code
```iecst
PROGRAM _INIT

	//Enable ImportAllowed
	MpIOImport_0.ImportAllowed := TRUE;

END_PROGRAM
PROGRAM _CYCLIC

	FileName := MpIOImportUIConnect.FileList.Names[MpIOImportUIConnect.FileList.Scroll.SelectedIndex];
	ActiveConfiguration;

	//Set FB parameters
	MpIOImport_0(
		Enable := TRUE,
		MpLink := ADR(gIoConfig),
		DeviceName := ADR('mappIO'),
		FileName := ADR(FileName));

	MpIOImportUI_0(
		Enable := TRUE,
		MpLink := ADR(gIoConfig),
		UIConnect := ADR(MpIOImportUIConnect));

	//Reset Import command if import succeded
	IF MpIOImport_0.CommandDone = TRUE THEN
		MpIOImport_0.Import := FALSE;
	END_IF

END_PROGRAM
PROGRAM _EXIT

	//Disable FBs
	MpIOImport_0(Enable := FALSE, ImportAllowed := FALSE);
	MpIOImportUI_0(Enable := FALSE);

END_PROGRAM
```

#### Variables.var - Local variables
```iecst
VAR
	FileName : STRING[80] := ''; (*FileName of HWConfig file*)
	MpIOImportUIConnect : MpIOImportUIConnectType;
	MpIOImportUI_0 : MpIOImportUI;
	MpIOImport_0 : MpIOImport;
	ActiveConfiguration : STRING[80] := 'Configuration 1';
END_VAR
```

### Program Logical/Infrastructure/Sequence (IEC) - Sequencer handling

#### Types.typ
```iecst
TYPE
	TONType : 	STRUCT
		AxisLeft : TON := (PT:=T#3S);
		TakeOutCup : TON := (PT:=T#3S);
		Coffee : TON := (PT:=T#3S);
		AxisRight : TON := (PT:=T#3S);
		Wait : TON := (PT:=T#3S);
		Start : TON := (PT:=T#1S);
		Stop : TON := (PT:=T#1S);
		ExecuteWait : TON := (PT:=T#2S);
		StopButton : TON;
		CoffeeWait : TON;
	END_STRUCT;
	SequencerStateEnum :
		(
		IDLE,
		MOVE_AXIS_LEFT,
		MOVE_AXIS_RIGHT,
		WAIT,
		COFFEE,
		STOP,
		TAKE_OUT,
		START
		);
	SequencerCommandType : 	STRUCT
		AxisLeft : MpSequencerCommandType;
		Stop : MpSequencerCommandType;
		TakeOutCup : MpSequencerCommandType;
		Coffee : MpSequencerCommandType;
		AxisRight : MpSequencerCommandType;
		Wait : MpSequencerCommandType;
		Start : MpSequencerCommandType;
		End : MpSequencerCommandType;
	END_STRUCT;
END_TYPE
```

#### Variables.var
```iecst
VAR
	Transform : STRING[1000] := '0';
	Timer : TONType := (0);
	SequenceStart : BOOL := 0;
	SavePressed : BOOL := FALSE;
	ParametersCore : MpSequenceCoreParType; (*Parameters for Core function block*)
	MpSequenceCore_0 : MpSequenceCore; (*Inizialize SequencCore function block*)
	EditSequence : BOOL := 0;
	CmdSeq : SequencerCommandType := (0); (*commandstructure for movement command Coffee*)
END_VAR
```

#### Main.st
```iecst
PROGRAM _INIT

	//Enable FBs and set parameters
	MpSequenceCore_0.Enable := TRUE;
	MpSequenceCore_0.Import := TRUE;
	MpSequenceCore_0.Mode := mpSEQUENCE_MODE_SINGLE_CYCLE;
	ParametersCore.Sequence := 'CoffeeSequence.xml';

	Timer.AxisLeft.PT := T#03s;
	Timer.AxisRight.PT := T#03s;
	Timer.Coffee.PT := T#03s;
	Timer.ExecuteWait.PT := T#03s;
	Timer.Start.PT := T#500ms;
	Timer.Stop.PT := T#01s;
	Timer.TakeOutCup.PT := T#01s;
	Timer.Wait.PT := T#03s;
	Timer.StopButton.PT := T#02s;
	Timer.CoffeeWait.PT := T#01s;

END_PROGRAM
PROGRAM _CYCLIC

	//Set FB parameters
	MpSequenceCore_0.MpLink := ADR(gSequenceCore);
	MpSequenceCore_0.Parameters := ADR(ParametersCore);

	IF MpSequenceCore_0.ImportDone THEN
		MpSequenceCore_0.Import := FALSE;
	END_IF

	//Start if Start-Button is pressed
	IF SequenceStart AND MpSequenceCore_0.Info.ReadyToStart THEN
		MpSequenceCore_0.Start := TRUE;
		EditSequence := FALSE;
		MpSequenceCore_0.ErrorReset := FALSE;
	ELSE

		MpSequenceCore_0.Start := FALSE;
		CmdSeq.Start.MovementState := mpSEQUENCE_MOVEMENT_IDLE;
		CmdSeq.AxisLeft.MovementState := mpSEQUENCE_MOVEMENT_IDLE;
		CmdSeq.AxisRight.MovementState := mpSEQUENCE_MOVEMENT_IDLE;
		CmdSeq.Coffee.MovementState := mpSEQUENCE_MOVEMENT_IDLE;
		CmdSeq.End.MovementState := mpSEQUENCE_MOVEMENT_IDLE;
		CmdSeq.TakeOutCup.MovementState := mpSEQUENCE_MOVEMENT_IDLE;
		CmdSeq.Wait.MovementState := mpSEQUENCE_MOVEMENT_IDLE;
		Timer.AxisLeft.IN := FALSE;
		Timer.AxisRight.IN := FALSE;
		Timer.Coffee.IN := FALSE;
		Timer.ExecuteWait.IN := FALSE;
		Timer.Start.IN := FALSE;
		Timer.Stop.IN := FALSE;
		Timer.TakeOutCup.IN := FALSE;
		Timer.Wait.IN := FALSE;
		Timer.StopButton.IN := TRUE;

		Transform := '[{"select":"#g83","duration":1000,"translate":[3.497,-208.81101],"display":true}
		,{"select":"#rect999-9-2","duration":1000,"display":false}
		,{"select":"#rect999-1","duration":1000,"display":false}
		,{"select":"#path49","duration":2000,"fill":7}
		,{"select":"#path39","duration":2000,"fill":0}
		,{"select":"#path41","duration":2000,"fill":2}
		,{"select":"#path3","duration":2000,"fill":3}
		,{"select":"#gLamp1","duration":2000,"fill":7}
		,{"select":"#gLamp2","duration":2000,"fill":7}
		,{"select":"#gLamp3","duration":2000,"fill":7}
		,{"select":"#gLamp4","duration":2000,"fill":7}
		,{"select":"#gLamp5","duration":2000,"fill":7}
		,{"select":"#gLamp6","duration":2000,"fill":7}]';

		IF Timer.StopButton.Q THEN
			Timer.StopButton.IN := FALSE;
		END_IF

		EditSequence := TRUE;

	END_IF

	(****************************************************************START*********************************************************************)
	IF CmdSeq.Start.Start THEN

		CmdSeq.Start.MovementState := mpSEQUENCE_MOVEMENT_ACTIVE;
		Timer.Start.IN := TRUE;
		Transform := '[{"select":"#g83","duration":500,"display":true}]';
		IF Timer.Start.Q THEN
			Timer.Start.IN := FALSE;
			CmdSeq.Start.MovementState := mpSEQUENCE_MOVEMENT_DONE;
		END_IF

	ELSE
		CmdSeq.Start.MovementState := mpSEQUENCE_MOVEMENT_IDLE;
	END_IF

	(****************************************************************AXIS LEFT*********************************************************************)
	IF CmdSeq.AxisLeft.Start THEN

		CmdSeq.AxisLeft.MovementState := mpSEQUENCE_MOVEMENT_ACTIVE;
		Timer.AxisLeft.IN := TRUE;
		Transform := '[{"select":"#g83","duration":3000,"translate":[440,-208.81101]},{"select":"#gLamp1","duration":2000,"fill":8},{"select":"#gLamp4","duration":2000,"fill":8}]';
		IF Timer.AxisLeft.Q THEN
			Timer.AxisLeft.IN := FALSE;
			CmdSeq.AxisLeft.MovementState := mpSEQUENCE_MOVEMENT_DONE;
		END_IF
	ELSE
		CmdSeq.AxisLeft.MovementState := mpSEQUENCE_MOVEMENT_IDLE;
	END_IF

	(****************************************************************AXIS RIGHT*********************************************************************)
	IF CmdSeq.AxisRight.Start THEN

		CmdSeq.AxisRight.MovementState := mpSEQUENCE_MOVEMENT_ACTIVE;
		Timer.AxisRight.IN := TRUE;
		Transform := '[{"select":"#g83","duration":3000,"translate":[560,-208.81101]},{"select":"#gLamp3","duration":2000,"fill":10},{"select":"#gLamp6","duration":2000,"fill":10}]';
		IF Timer.AxisRight.Q THEN
			Timer.AxisRight.IN := FALSE;
			CmdSeq.AxisRight.MovementState := mpSEQUENCE_MOVEMENT_DONE;
		END_IF
	ELSE
		CmdSeq.AxisRight.MovementState := mpSEQUENCE_MOVEMENT_IDLE;
	END_IF

	(****************************************************************COFFEE*********************************************************************)
	IF CmdSeq.Coffee.Start THEN

		CmdSeq.Coffee.MovementState := mpSEQUENCE_MOVEMENT_ACTIVE;
		Timer.Coffee.IN := TRUE;
		Transform :='[{"select":"#path39","duration":2000,"fill":7}
		,{"select":"#path41","duration":2000,"fill":7}
		,{"select":"#path3","duration":2000,"fill":7}
		,{"select":"#gLamp2","duration":2000,"fill":9},
		{"select":"#gLamp5","duration":2000,"fill":9}]';
		IF Timer.Coffee.Q THEN

			Timer.ExecuteWait.IN := TRUE;

			Transform := '[{"select":"#rect999-9-2","duration":2000,"display":true,"fill":1}
			,{"select":"#rect999-1","duration":2000,"display":true,"fill":1}
			,{"select":"#path49","duration":2000,"fill":0}
			,{"select":"#path39","duration":2000,"fill":0}
			,{"select":"#path41","duration":2000,"fill":2}
			,{"select":"#path3","duration":2000,"fill":3}]';
			IF Timer.ExecuteWait.Q THEN

				Timer.CoffeeWait.IN := TRUE;
				Transform := '[{"select":"#rect999-1","duration":1000,"display":false},
				{"select":"#rect999-9-2","duration":1000,"display":false},
				{"select":"#path49","duration":1000,"fill":7}]';
				IF Timer.CoffeeWait.Q THEN
					Timer.CoffeeWait.IN := FALSE;
					Timer.Coffee.IN := FALSE;
					Timer.ExecuteWait.IN := FALSE;
					CmdSeq.Coffee.MovementState := mpSEQUENCE_MOVEMENT_DONE;
				END_IF
			END_IF
		END_IF

	ELSE
		CmdSeq.Coffee.MovementState := mpSEQUENCE_MOVEMENT_IDLE;
	END_IF

	(****************************************************************TAKEOUT*********************************************************************)
	IF CmdSeq.TakeOutCup.Start THEN

		CmdSeq.TakeOutCup.MovementState := mpSEQUENCE_MOVEMENT_ACTIVE;
		Timer.TakeOutCup.IN := TRUE;
		Transform := '[{"select":"#g83","duration":500,"display":false}]';
		IF Timer.TakeOutCup.Q THEN
			Timer.TakeOutCup.IN := FALSE;
			CmdSeq.TakeOutCup.MovementState := mpSEQUENCE_MOVEMENT_DONE;
		END_IF
	ELSE
		CmdSeq.TakeOutCup.MovementState := mpSEQUENCE_MOVEMENT_IDLE;
	END_IF

	(****************************************************************WAIT*********************************************************************)
	IF CmdSeq.Wait.Start THEN
		CmdSeq.Wait.MovementState := mpSEQUENCE_MOVEMENT_ACTIVE;
		Timer.Wait.IN := TRUE;

		IF Timer.Wait.Q THEN
			Timer.Wait.IN := FALSE;
			CmdSeq.Wait.MovementState := mpSEQUENCE_MOVEMENT_DONE;
		END_IF
	ELSE
		CmdSeq.Wait.MovementState := mpSEQUENCE_MOVEMENT_IDLE;
	END_IF

	(****************************************************************STOP*********************************************************************)
	IF CmdSeq.Stop.Start THEN
		CmdSeq.Stop.MovementState := mpSEQUENCE_MOVEMENT_ACTIVE;
		Timer.Stop.IN := TRUE;
		Transform := '[{"select":"#g83","duration":1000,"translate":[3.497,-208.81101]}
		]';

		IF Timer.Stop.Q THEN
			Timer.Stop.IN := FALSE;
			CmdSeq.Stop.MovementState := mpSEQUENCE_MOVEMENT_DONE;
			Transform := '[{"select":"#g83","duration":500,"display":true}]';
			SequenceStart := FALSE;
		END_IF
	ELSE
		CmdSeq.Stop.MovementState := mpSEQUENCE_MOVEMENT_IDLE;
	END_IF

	(****************************************************************ERROR*********************************************************************)
	IF MpSequenceCore_0.Error THEN
		SequenceStart := FALSE;
		MpSequenceCore_0.Import := FALSE;
		MpSequenceCore_0.ErrorReset := gCoffeeMainLogic.cmdClear;
	END_IF

	IF SavePressed THEN
		MpSequenceCore_0.Import := TRUE;
		SavePressed := FALSE;
	END_IF

	//Call FB
	MpSequenceCore_0();
	Timer.AxisLeft();
	Timer.AxisRight();
	Timer.Coffee();
	Timer.Start();
	Timer.Stop();
	Timer.TakeOutCup();
	Timer.Wait();
	Timer.ExecuteWait();
	Timer.StopButton();
	Timer.CoffeeWait();

END_PROGRAM
PROGRAM _EXIT

	//Disable FB
	MpSequenceCore_0(Enable := FALSE);

END_PROGRAM
```

### Program Logical/Infrastructure/CodeBox (IEC) - CodeBox handling

#### Main.st - Init, cyclic, exit code
```iecst
PROGRAM _INIT

	State := WAIT;

END_PROGRAM

PROGRAM _CYCLIC

	//Set FB parameter
	MpCodeBoxCore_0(
	MpLink := ADR(gCodeBoxCore),
	Enable := TRUE,
	ErrorReset := gCoffeeMainLogic.cmdClear);

	Cup;
	Lamp;

	CodeBoxTransform;

	CASE State OF
		WAIT:
			CodeBoxTransform := '[{"select":"#gLamp1","duration":200,"fill":7}
			,{"select":"#gLamp2","duration":200,"fill":7}
			,{"select":"#gLamp3","duration":200,"fill":7}
			,{"select":"#gLamp4","duration":200,"fill":7}
			,{"select":"#gLamp5","duration":200,"fill":7}
			,{"select":"#gLamp6","duration":200,"fill":7}]';

			IF gCoffeeMainLogic.PackMLState = 'Idle' THEN
				State := CUP_START_POS;

			END_IF

		CUP_START_POS:
			Cup.StartPosition := TRUE;
			IF Lamp.Green THEN

				CodeBoxTransform := '[{"select":"#gLamp1","duration":1000,"fill":10}
					,{"select":"#gLamp2","duration":1000,"fill":7}
					,{"select":"#gLamp3","duration":1000,"fill":7}
					,{"select":"#gLamp4","duration":1000,"fill":10}
					,{"select":"#gLamp5","duration":1000,"fill":7}
					,{"select":"#gLamp6","duration":1000,"fill":7}]';

			ELSIF Lamp.Red THEN
				CodeBoxTransform := '[{"select":"#gLamp1","duration":1000,"fill":8}
				,{"select":"#gLamp2","duration":1000,"fill":7}
				,{"select":"#gLamp3","duration":1000,"fill":7}
				,{"select":"#gLamp4","duration":1000,"fill":8}
				,{"select":"#gLamp5","duration":1000,"fill":7}
				,{"select":"#gLamp6","duration":1000,"fill":7}]';

			ELSIF Lamp.Yellow THEN
				CodeBoxTransform := '[{"select":"#gLamp1","duration":1000,"fill":9}
				,{"select":"#gLamp2","duration":1000,"fill":7}
				,{"select":"#gLamp3","duration":1000,"fill":7}
				,{"select":"#gLamp4","duration":1000,"fill":9}
				,{"select":"#gLamp5","duration":1000,"fill":7}
				,{"select":"#gLamp6","duration":1000,"fill":7}]';
			ELSE
				CodeBoxTransform := '[{"select":"#gLamp1","duration":1000,"fill":7}
				,{"select":"#gLamp2","duration":1000,"fill":7}
				,{"select":"#gLamp3","duration":1000,"fill":7}
				,{"select":"#gLamp4","duration":1000,"fill":7}
				,{"select":"#gLamp5","duration":1000,"fill":7}
				,{"select":"#gLamp6","duration":1000,"fill":7}]';
			END_IF

			IF gCoffeeMainLogic.PackMLState = 'Execute' THEN
				State := CUP_COFFEE;
				Cup.StartPosition := FALSE;
			END_IF

		CUP_COFFEE:
			Cup.CoffeePosition := TRUE;
			IF gCoffeeMainLogic.PackMLState = 'Completing' THEN
				State := CUP_END_POS;
				Cup.CoffeePosition := FALSE;
			END_IF

			IF Lamp.Green THEN

				CodeBoxTransform := '[{"select":"#gLamp1","duration":1000,"fill":7}
				,{"select":"#gLamp2","duration":1000,"fill":10}
				,{"select":"#gLamp3","duration":1000,"fill":7}
				,{"select":"#gLamp4","duration":1000,"fill":7}
				,{"select":"#gLamp5","duration":1000,"fill":10}
				,{"select":"#gLamp6","duration":1000,"fill":7}]';

			ELSIF Lamp.Red THEN
				CodeBoxTransform := '[{"select":"#gLamp1","duration":1000,"fill":7}
				,{"select":"#gLamp2","duration":1000,"fill":8}
				,{"select":"#gLamp3","duration":1000,"fill":7}
				,{"select":"#gLamp4","duration":1000,"fill":7}
				,{"select":"#gLamp5","duration":1000,"fill":8}
				,{"select":"#gLamp6","duration":1000,"fill":7}]';

			ELSIF Lamp.Yellow THEN
				CodeBoxTransform := '[{"select":"#gLamp1","duration":1000,"fill":7}
				,{"select":"#gLamp2","duration":1000,"fill":9}
				,{"select":"#gLamp3","duration":1000,"fill":7}
				,{"select":"#gLamp4","duration":1000,"fill":7}
				,{"select":"#gLamp5","duration":1000,"fill":9}
				,{"select":"#gLamp6","duration":1000,"fill":7}]';
			ELSE
				CodeBoxTransform := '[{"select":"#gLamp1","duration":1000,"fill":7}
				,{"select":"#gLamp2","duration":1000,"fill":7}
				,{"select":"#gLamp3","duration":1000,"fill":7}
				,{"select":"#gLamp4","duration":1000,"fill":7}
				,{"select":"#gLamp5","duration":1000,"fill":7}
				,{"select":"#gLamp6","duration":1000,"fill":7}]';
			END_IF
		CUP_END_POS:
			Cup.EndPosition := TRUE;
			IF Lamp.Green THEN

				CodeBoxTransform := '[{"select":"#gLamp1","duration":1000,"fill":7}
				,{"select":"#gLamp2","duration":1000,"fill":7}
				,{"select":"#gLamp3","duration":1000,"fill":10}
				,{"select":"#gLamp4","duration":1000,"fill":7}
				,{"select":"#gLamp5","duration":1000,"fill":7}
				,{"select":"#gLamp6","duration":1000,"fill":10}]';

			ELSIF Lamp.Red THEN
				CodeBoxTransform := '[{"select":"#gLamp1","duration":1000,"fill":7}
				,{"select":"#gLamp2","duration":1000,"fill":7}
				,{"select":"#gLamp3","duration":1000,"fill":8}
				,{"select":"#gLamp4","duration":1000,"fill":7}
				,{"select":"#gLamp5","duration":1000,"fill":7}
				,{"select":"#gLamp6","duration":1000,"fill":8}]';

			ELSIF Lamp.Yellow THEN
				CodeBoxTransform := '[{"select":"#gLamp1","duration":1000,"fill":7}
				,{"select":"#gLamp2","duration":1000,"fill":7}
				,{"select":"#gLamp3","duration":1000,"fill":9}
				,{"select":"#gLamp4","duration":1000,"fill":7}
				,{"select":"#gLamp5","duration":1000,"fill":7}
				,{"select":"#gLamp6","duration":1000,"fill":9}]';
			ELSE
				CodeBoxTransform := '[{"select":"#gLamp1","duration":1000,"fill":7}
				,{"select":"#gLamp2","duration":1000,"fill":7}
				,{"select":"#gLamp3","duration":1000,"fill":7}
				,{"select":"#gLamp4","duration":1000,"fill":7}
				,{"select":"#gLamp5","duration":1000,"fill":7}
				,{"select":"#gLamp6","duration":1000,"fill":7}]';
			END_IF
			IF gCoffeeMainLogic.PackMLState = 'Idle' THEN
				State := WAIT;
				Cup.EndPosition := FALSE;
			END_IF

	END_CASE

END_PROGRAM

PROGRAM _EXIT

	MpCodeBoxCore_0(Enable := FALSE);

END_PROGRAM
```

#### Types.typ - Local data types
```iecst
TYPE
	CodeBox_State :
		(
		WAIT := 0,
		CUP_COFFEE := 1,
		CUP_END_POS := 2,
		CUP_START_POS := 3
		);
	Cup_Type : 	STRUCT
		StartPosition : BOOL;
		EndPosition : BOOL;
		CoffeePosition : BOOL;
	END_STRUCT;
	Lamp_type : 	STRUCT
		Red : BOOL;
		Yellow : BOOL;
		Green : BOOL;
	END_STRUCT;
END_TYPE
```

#### Variables.var - Local variables
```iecst
VAR
	State : CodeBox_State := CUP_START_POS;
	Cup : Cup_Type := (0);
	MpCodeBoxCore_0 : MpCodeBoxCore := (0);
	Lamp : Lamp_type := (0);
	CodeBoxTransform : STRING[2000] := '';
END_VAR
```

- Project.language (not shown)

### Package Logical/Industry - Industry Components

### Program Logical/Industry/PackML (IEC) - PackML handling

#### Variables.var
```iecst
VAR
	MpPackMLBasicUI_0 : MpPackMLBasicUI; (*MpPackMLBasicUI instance*)
	MpPackMLBasicUIConnect : MpPackMLBasicUIConnectType := (ModeControl:=(SelectedIndex:=1)); (*MpPackMLBasicUI UI connection datapoints*)
	MpPackMLStatisticsUI_0 : MpPackMLStatisticsUI; (*MpPackMLStatisticsUI instance*)
	MpPackMLStatisticsUIConnect : MpPackMLStatisticsUIConnectType; (*MpPackMLStatistics UI connection datapoints*)
	MpPackMLMode_0 : MpPackMLMode;
	MpPackMLCore_0 : MpPackMLCore;
	MpPackMLMode_1 : MpPackMLMode;
END_VAR
```

#### Main.st
```iecst
PROGRAM _CYCLIC

	//Set FB parameters
	MpPackMLCore_0(
		MpLink := ADR(gPackMLCore),
		Enable := TRUE);

	MpPackMLMode_0(
		MpLink := ADR(gPackMLCore),
		Enable := TRUE,
		ModeID := PACKML_MODE_PRODUCTION,
		Start := gCoffeeMainLogic.cmdStart,
		Stop := gCoffeeMainLogic.cmdStop,
		Reset := MpPackMLStateIsActive(gPackMLCore,mpPACKML_STATE_STOPPED,PACKML_MODE_PRODUCTION),
		Abort := (gCoffeeMainLogic.cmdAbort AND MpPackMLMode_0.ModeActive),
		Clear := gCoffeeMainLogic.cmdClear);

	MpPackMLMode_1(
		MpLink := ADR(gPackMLCore),
		Enable := TRUE,
		ModeID := PACKML_MODE_MAINTENANCE);

	MpPackMLBasicUI_0(
		MpLink := ADR(gPackMLCore),
		Enable := TRUE,
		UIConnect := ADR(MpPackMLBasicUIConnect));

	MpPackMLStatisticsUI_0(
		MpLink := ADR(gPackMLCore),
		Enable := TRUE,
		UIConnect := ADR(MpPackMLStatisticsUIConnect));

	//Check if you can refill the ingredients
	IF MpPackMLCore_0.Info.StateCurrent = 'Idle' OR MpPackMLCore_0.Info.StateCurrent = 'Aborted' THEN
		gCoffeeMainLogic.IdleState := TRUE;
	ELSE
		gCoffeeMainLogic.IdleState := FALSE;
	END_IF

END_PROGRAM
PROGRAM _EXIT

	//Disable FBs
	MpPackMLCore_0(Enable := FALSE);
	MpPackMLMode_0(Enable := FALSE);
	MpPackMLMode_1(Enable := FALSE);
	MpPackMLBasicUI_0(Enable := FALSE);
	MpPackMLStatisticsUI_0(Enable := FALSE);

END_PROGRAM
```

### Program Logical/MainControl (IEC) - MainContol program

#### Cyclic.st - Cyclic code
```iecst
PROGRAM _CYCLIC

	// Main state machine for the brewing process handled by PackML

(****************************************************************IDLE*********************************************************************)

	IF (MpPackMLStateIsActive(gPackMLCore, mpPACKML_STATE_IDLE, PACKML_MODE_PRODUCTION)) THEN
		gCoffeeMainLogic.PackMLState := 'Idle';
		TransitionTime := 500;
		TransformTime := T#500ms;
		gCoffeeMainLogic.AxisCupFeeder.Power 		:= TRUE;
		gCoffeeMainLogic.AxisTakeout.Power 			:= TRUE;

		IF (gCoffeeMainLogic.AxisTakeout.Active = TRUE) AND (gCoffeeMainLogic.AxisCupFeeder.Active = TRUE)  THEN

			MainCoffeeUIConnect.visShowButtonStart 	:= YES;
			MainCoffeeUIConnect.visWaterLevel 		:= 100;	// initialize water level
			Transform := '[{"select":"#g83","duration":500,"display":true}]';
		ELSE

			gCoffeeMainLogic.cmdAbort := TRUE;

		END_IF

	END_IF

	(****************************************************************RESETTING*********************************************************************)

	IF (MpPackMLStateIsActive(gPackMLCore, mpPACKML_STATE_RESETTING
		, PACKML_MODE_PRODUCTION)) THEN
		gCoffeeMainLogic.PackMLState := 'Resetting';
		gCoffeeMainLogic.cmdClear 		:= FALSE;
		gCoffeeMainLogic.cmdAbort 		:= FALSE;

		gCoffeeMainLogic.AxisCupFeeder.Power 		:= TRUE;				// power and home both conveyor axes
		gCoffeeMainLogic.AxisTakeout.Power 			:= TRUE;

		IF(gCoffeeMainLogic.AxisTakeout.PowerOn = TRUE) AND (gCoffeeMainLogic.AxisCupFeeder.PowerOn = TRUE)  THEN

			MpPackMLStateComplete(gPackMLCore, PACKML_MODE_PRODUCTION);

		END_IF
	END_IF

	(******************************************************************STARTING*******************************************************************)

	IF (MpPackMLStateIsActive(gPackMLCore, mpPACKML_STATE_STARTING, PACKML_MODE_PRODUCTION)) THEN
		gCoffeeMainLogic.PackMLState := 'Starting';
		MainCoffeeUIConnect.visShowMainBrewing 			:= YES;
		MainCoffeeUIConnect.visShowMainRecipe  			:= YES;
		MainCoffeeUIConnect.visShowButtonStart 			:= NO;
		MainCoffeeUIConnect.visCupSlider 				:= 0;

		TransitionTime := 3000;
		Transform := '[{"select":"#g83","duration":3000,"translate":[375,-87.299533]}]';
		TransformTime := T#3S;
		TransformWait.IN := TRUE;
		TransformWait.PT := TransformTime;

		gCoffeeMainLogic.AxisCupFeeder.MoveAdditive 	:= TRUE;			// start moving the cup to fill station
		gCoffeeMainLogic.cmdStart := FALSE;

		IF (gCoffeeMainLogic.AxisCupFeeder.InPosition) AND TransformWait.Q = TRUE THEN
			TransformWait.IN := FALSE;
			gCoffeeMainLogic.AxisCupFeeder.MoveAdditive 	:= FALSE;				// reset command when in position
			MainCoffeeUIConnect.visCupSlider 				:= 1000;
			gCoffeeMainLogic.AxisCupFeeder.InPosition := FALSE;
			gCoffeeMainLogic.AxisCupFeeder.Position 	:= 0.0;
			MpPackMLStateComplete(gPackMLCore, PACKML_MODE_PRODUCTION);
			TransformWait();
		END_IF

	END_IF

	(******************************************************************EXECUTE*******************************************************************)

	IF (MpPackMLStateIsActive(gPackMLCore, mpPACKML_STATE_EXECUTE, PACKML_MODE_PRODUCTION)) THEN
		gCoffeeMainLogic.PackMLState := 'Execute';
		TransitionTime := 3000;
		TransformTime := T#3S;
		Transform :='[{"select":"#path39","duration":2000,"fill":7}
		,{"select":"#path41","duration":2000,"fill":7}
		,{"select":"#path3","duration":2000,"fill":7}
		,{"select":"#rect999","duration":2000,"display":true,"fill":1}
		,{"select":"#rect999-9","duration":2000,"display":true,"fill":1}
		,{"select":"#path49","duration":2000,"fill":0}]';
		ExecuteWait.IN := TRUE;
		ExecuteWait.PT := TransformTime;
		ExecuteWait();

		IF ExecuteWait.Q = TRUE THEN
			FillCoffeeWait.IN := TRUE;
			FillCoffeeWait.PT := T#2s;
			Transform := '[{"select":"#path49","duration":2000,"fill":0}
			,{"select":"#path39","duration":2000,"fill":0}
			,{"select":"#path41","duration":2000,"fill":2}
			,{"select":"#path3","duration":2000,"fill":3}
			,{"select":"#rect999","duration":500,"display":false}
			,{"select":"#rect999-9","duration":500,"display":false}
			,{"select":"#path49","duration":2000,"fill":7}]';

			IF FillCoffeeWait.Q THEN
				FillCoffeeWait.IN := FALSE;
				ExecuteWait.IN := FALSE;
				gCoffeeMainLogic.AxisTakeout.MoveAdditive := TRUE;					// start moving cup to take out
				MpPackMLStateComplete(gPackMLCore, PACKML_MODE_PRODUCTION);
			END_IF
		END_IF

	END_IF

	(******************************************************************Completing*******************************************************************)

	IF (MpPackMLStateIsActive(gPackMLCore, mpPACKML_STATE_COMPLETING, PACKML_MODE_PRODUCTION)) THEN
		TransitionTime := 3000;
		Transform := '[{"select":"#g83","duration":3000,"translate":[560,-87.299533]}]';
		gCoffeeMainLogic.PackMLState := 'Completing';
		TransformWait.IN := TRUE;
		TransformWait.PT := TransformTime;

		IF (gCoffeeMainLogic.AxisTakeout.InPosition) AND TransformWait.Q = TRUE THEN

			TransitionTime := 500;
			Transform := '[{"select":"#g83","duration":500,"display":false}]';
			TransformHide.IN := TRUE;
			TransformHide.PT := TransformTime;

			IF TransformHide.Q = TRUE THEN

				CupHideWait.IN := TRUE;
				CupHideWait.PT := T#1S;
				Transform := '[{"select":"#g83","duration":1000,"translate":[3.497,-87.299533]}]';

				IF CupHideWait.Q = TRUE THEN
					CupHideWait.IN := FALSE;
					TransformWait.IN := FALSE;
					TransformHide.IN := FALSE;
					MainCoffeeUIConnect.visShowMainBrewing 		:= NO;
					MainCoffeeUIConnect.visShowMainRecipe  		:= NO;
					MainCoffeeUIConnect.visCupSlider 			:= 2000;
					gCoffeeMainLogic.cmdStart					:= FALSE;					// reset the brewing start command
					gCoffeeMainLogic.AxisTakeout.MoveAdditive 	:= FALSE;					// reset command when in position
					gCoffeeMainLogic.AxisTakeout.InPosition := FALSE;
					gCoffeeMainLogic.AxisTakeout.Position 	:= 0.0;
					MpPackMLStateComplete(gPackMLCore, PACKML_MODE_PRODUCTION);
				END_IF

			END_IF

		END_IF

	END_IF
	TransformWait();
	CupHideWait();
	TransformHide();
	(****************************************************************STOPPED*********************************************************************)

	IF (MpPackMLStateIsActive(gPackMLCore, mpPACKML_STATE_STOPPED, PACKML_MODE_PRODUCTION)) THEN
		gCoffeeMainLogic.PackMLState := 'Stopped';
		gCoffeeMainLogic.cmdClear := FALSE;
		MainCoffeeUIConnect.visShowAlarmBanner 	:= NO;

	END_IF

	(******************************************************************ABORTING*******************************************************************)

	IF (MpPackMLStateIsActive(gPackMLCore, mpPACKML_STATE_ABORTING, PACKML_MODE_PRODUCTION)) THEN
		gCoffeeMainLogic.PackMLState := 'Aborting';
		MainCoffeeUIConnect.visShowButtonStart 	:= NO;
		MainCoffeeUIConnect.visShowMainBrewing 	:= NO;
		MainCoffeeUIConnect.visShowMainRecipe  	:= NO;
		MainCoffeeUIConnect.visShowAlarmBanner 	:= YES;
		MainCoffeeUIConnect.visShowButtonStart 	:= NO;

		gCoffeeMainLogic.AxisCupFeeder.Power 	:= FALSE;
		gCoffeeMainLogic.AxisTakeout.Power 		:= FALSE;

		IF (gCoffeeMainLogic.AxisCupFeeder.PowerOn = FALSE) AND (gCoffeeMainLogic.AxisTakeout.PowerOn = FALSE) THEN
			MpPackMLStateComplete(gPackMLCore, PACKML_MODE_PRODUCTION);
		END_IF

		gCoffeeMainLogic.cmdAbort := FALSE;
	END_IF

	(******************************************************************ABORTED*******************************************************************)

	IF (MpPackMLStateIsActive(gPackMLCore, mpPACKML_STATE_ABORTED, PACKML_MODE_PRODUCTION)) THEN
		gCoffeeMainLogic.PackMLState := 'Aborted';
		gCoffeeMainLogic.AxisCupFeeder.Power 			:= FALSE;
		gCoffeeMainLogic.AxisTakeout.Power 				:= FALSE;
		gCoffeeMainLogic.AxisCupFeeder.MoveAdditive 	:= FALSE;
		gCoffeeMainLogic.AxisTakeout.MoveAdditive		:= FALSE;
		gCoffeeMainLogic.AxisCupFeeder.Home			 	:= FALSE;
		gCoffeeMainLogic.AxisTakeout.Home				:= FALSE;

		IF (gCoffeeMainLogic.AxisCupFeeder.PowerOn = FALSE) AND (gCoffeeMainLogic.AxisTakeout.PowerOn = FALSE) THEN
			MpPackMLStateComplete(gPackMLCore, PACKML_MODE_PRODUCTION);
		END_IF

		gCoffeeMainLogic.cmdAbort := FALSE;
	END_IF

	(******************************************************************END OF PACKML*******************************************************************)

	RecipeRegister;
	UserLevelCheck;

	//Check if Alarm can be cleared
	IF (gClearAlarm = TRUE) THEN
		MainCoffeeUIConnect.visShowClearButton := YES;
	ELSE
		MainCoffeeUIConnect.visShowClearButton := NO;
	END_IF

	//Control Refill Alarms
	IF MainCoffeeUIConnect.visStartCoffee = TRUE THEN
		gCoffeeMainLogic.cmdStart := TRUE;
		(*gCoffeeMainLogic.cmdClear := TRUE*)
		MainCoffeeUIConnect.visStartCoffee := FALSE;
		ProducedCoffee.Number := ProducedCoffee.Number + 1;

		Refill.Coffee := Refill.Coffee - gCoffeeMainLogic.Refill.Coffee;
		Refill.Milk := Refill.Milk - gCoffeeMainLogic.Refill.Milk;
		Refill.Sugar := Refill.Sugar - gCoffeeMainLogic.Refill.Sugar;
		Refill.Water := Refill.Water - gCoffeeMainLogic.Refill.Water;

	END_IF

	TransformWait();
	FillCoffeeWait();
	ExecuteWait();
END_PROGRAM
```

#### Init.st
```iecst
PROGRAM _INIT
	MainCoffeeUIConnect.visCoffeeLevel := 100;
	MainCoffeeUIConnect.visMilkLevel := 100;
	MainCoffeeUIConnect.visSugarLevel := 100;
	MainCoffeeUIConnect.visWaterLevel := 100;

END_PROGRAM
```

#### Variables.var - Local variables
```iecst
VAR
	FillCoffeeWait : TON := (0);
	ProducedCoffee : ProducedCoffeeType := (0);
	MainCoffeeUIConnect : MainCoffeeUIConnectType := (visShowMainBrewing:=1,visShowMainRecipe:=1,visShowButtonStart:=0,visWaterLevel:=50); (*Control structure of main logic*)
	MpRecipeRegPar_0 : MpRecipeRegPar; (*Registration of a variable into the recipe system*)
END_VAR
VAR CONSTANT
	YES : BOOL := FALSE; (*Display an element on the visualization screen*)
	NO : BOOL := TRUE; (*Hide an element on the visualization screen*)
END_VAR
VAR
	Refill : RefillMainType := (Milk:=1000,Sugar:=1000,Coffee:=1000,Water:=1000);
	Transform : STRING[1000000] := ''; (*transforms the svg image in the coffee Visualization*)
	TransformTime : TIME := T#3S;
	TransformWait : TON := (0);
	TransitionTime : UINT := 3000;
	ExecuteWait : TON;
	CupHideWait : TON := (0);
	TransformHide : TON;
END_VAR
```

#### Types.typ - Local types
```iecst
TYPE
	ProducedCoffeeType : 	STRUCT
		Number : INT;
		_Number : INT;
		Name : STRING[80];
	END_STRUCT;
	RefillMainType : 	STRUCT
		Milk : INT; (*Whole amount of milk*)
		Sugar : INT; (*Whole amount of sugar*)
		Coffee : INT; (*Whole amount of coffee*)
		Water : INT; (*Whole amount of water*)
	END_STRUCT;
	RecipeSelectEnum :
		( (*Enumeration definition for recipe selection*)
		MAPP_REGULAR := 0,
		MAPP_MILKCOFFEE := 1,
		MAPP_ESSPRESSO := 2,
		MAPP_CAPPUCINO := 3,
		NO_SELECTION := 4
		);
	MainControlStepEnum :
		( (*Enumeration definition for main state machine*)
		STATE_IDLE,
		STATE_STARTING,
		STATE_EXECUTE,
		STATE_COMPLETING,
		STATE_TAKEOUT_CUP,
		STATE_POSITION_CUP
		);
	RefillStateEnum :
		( (*Enumeration definition for refill machine*)
		REFILL_NONE := 1,
		REFILL_WATER := 2,
		REFILL_MILK := 3,
		REFILL_COFFEE := 4,
		REFILL_SUGAR := 5
		);
	MainCoffeeUIConnectType : 	STRUCT  (*Main logic structure *)
		visShowMainBrewing : BOOL; (*HMI control bit*)
		visShowMainRecipe : BOOL; (*HMI control bit*)
		visShowButtonClear : BOOL; (*HMI control bit*)
		visShowButtonStart : BOOL; (*HMI control bit*)
		visShowUserLevelWarning : BOOL; (*HMI control bit*)
		visShowAlarmBanner : BOOL; (*HMI control bit*)
		visCupSlider : UINT; (*HMI control element*)
		visWaterLevel : INT; (*HMI control element*)
		visShowClearButton : BOOL; (*HMI control bit*)
		visShowButtonTakeout : BOOL; (*HMI control bit*)
		visMilkLevel : INT; (*HMI control element*)
		visSugarLevel : INT; (*HMI control element*)
		visShowRecipeSelection : BOOL; (*HMI control bit*)
		visCoffeeLevel : INT; (*HMI control element*)
		RecipeIsSelected : BOOL; (*HMI control bit*)
		visShowMinusSugar : BOOL; (*HMI control bit*)
		visShowPlusSugar : BOOL; (*HMI control bit*)
		visContinueButton : BOOL; (*HMI control bit*)
		visStartCoffee : BOOL; (*HMI control bit*)
	END_STRUCT;
END_TYPE
```

#### User.st - User level check
```iecst
// use the MpUserLevel function to read the current user level so that a warning is displayed if too low for recipe changes
ACTION UserLevelCheck:

	IF (MpUserXLevel(gUserXLogin) < 100) THEN
		MainCoffeeUIConnect.visShowUserLevelWarning := TRUE;
	ELSE
		MainCoffeeUIConnect.visShowUserLevelWarning := FALSE;
	END_IF

END_ACTION
```

#### Recipe.st - Register PV for recipe handling
```iecst
// registering the PictureIndex variable as additional parameter to be saved with the recipe parameters
ACTION RecipeRegister:

	MpRecipeRegPar_0(MpLink := ADR(gRecipeXml),
	Enable := TRUE,
	PVName := ADR('gCoffeeMainLogic.visPictureIndex'));

END_ACTION
```

### Program Logical/WaterHeater (IEC) - WaterHeater contol program

#### Cyclic.ld - Cyclic code
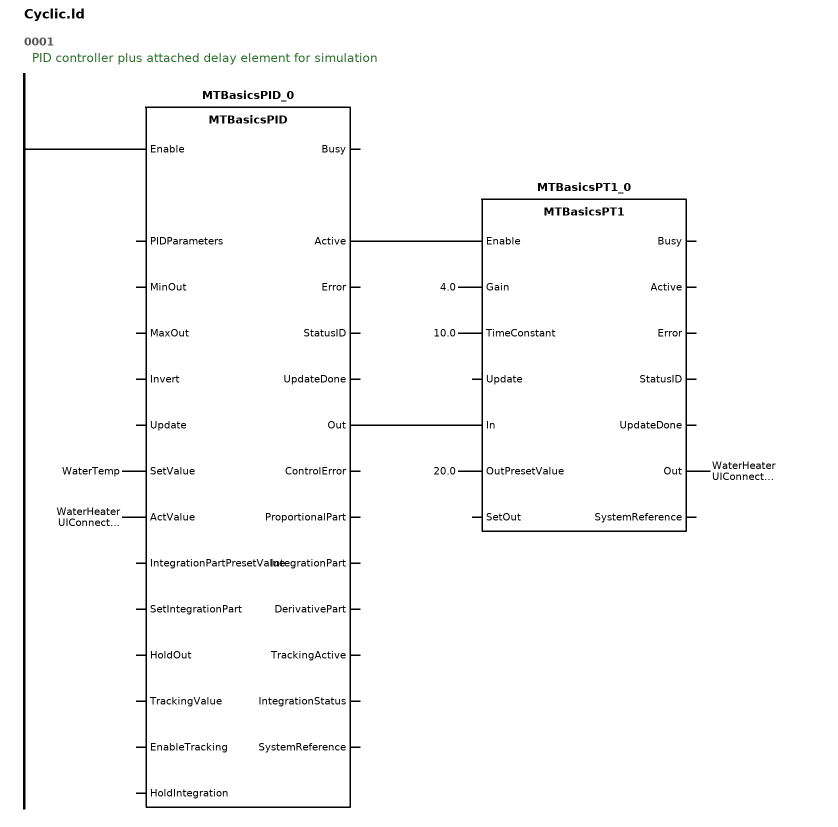
Ladder, written as Structured Text:
```iecst
PROGRAM _CYCLIC
(* Network 1: PID controller plus attached delay element for simulation *)
MTBasicsPID_0(Enable := TRUE, SetValue := WaterTemp, ActValue := WaterHeaterUIConnect.actTemperature);
MTBasicsPT1_0(Enable := MTBasicsPID_0.Active, Gain := 4.0, TimeConstant := 10.0, In := MTBasicsPID_0.Out, OutPresetValue := 20.0);
WaterHeaterUIConnect.actTemperature := MTBasicsPT1_0.Out;
END_PROGRAM
```

#### Variables.var - Local variables
```iecst
VAR
	MTBasicsPID_0 : MTBasicsPID := (PIDParameters:=(Gain:=4,IntegrationTime:=10),MinOut:=10,MaxOut:=100); (*MTBasicsPID instance*)
	MTBasicsPT1_0 : MTBasicsPT1; (*MTBasicsPT1 instance*)
	WaterTemp : REAL := 0.0; (*Water temperature for brewing coffee*)
	WaterHeaterUIConnect : WaterHeaterUIConnectType; (*Control structure of main logic*)
	MpEnergyRegPower_0 : MpEnergyRegPower := (0); (*MpEnergyRegPower instance*)
	MpEnergyRegEnergy_0 : MpEnergyRegEnergy := (0); (*MpEneryRegEnergy instance*)
	MpRecipeRegPar_0 : {REDUND_UNREPLICABLE} MpRecipeRegPar; (*MpRecipeRegPar instance*)

END_VAR
(*Variables for AuditTrail*)
VAR
	MpAuditValueChangeStatus : DINT; (*Status variable for MpAuditValueChange function*)
	_WaterTemp : REAL; (*Temp variables to detect value change*)
END_VAR
(*Variables for Energy monitoring*)
VAR
	ForwardActiveEnergy : LREAL := 0.0; (*Parameter for forward active energy*)
	ActivePower : LREAL := 0.0; (*Parameter for active power*)
END_VAR
```

#### Types.typ - Local types
```iecst
TYPE
	WaterHeaterUIConnectType : 	STRUCT  (*Main logic structure *)
		actTemperature : REAL; (*HMI actual temperature value*)
		setTemperature : REAL; (*HMI set temperature value*)
		visShowCooling : UINT; (*HMI control variable*)
		visShowHeating : UINT; (*HMI control variable*)
	END_STRUCT;
END_TYPE
```

#### Recipe.st - Register PV for recipe handling
```iecst
// registering the water temperature as additional parameter to be saved with the recipe parameters
ACTION RecipeRegister:

	MpRecipeRegPar_0(MpLink := ADR(gRecipeXml),
	Enable := TRUE,
	PVName := ADR('WaterHeater:WaterTemp'));

END_ACTION
```

#### Energy.st - Record energy usage for water heater
```iecst
ACTION Energy:
	ActivePower := 1800;
	ForwardActiveEnergy := MpEnergyRegEnergy_0.ForwardActiveEnergy + 0.1*ABS(MTBasicsPID_0.ControlError);

	MpEnergyRegPower_0(
		MpLink := ADR(gEnergyCore),
		Enable := TRUE,
		ModuleName := ADR('Waterheater Power'),
		Mode := mpENERGY_REG_MODE_COLLECT,
		Units := mpENERGY_POWER_UNIT_W,
		ActivePower := ActivePower);

	MpEnergyRegEnergy_0(
		MpLink := ADR(gEnergyCore),
		Enable := TRUE,
		ModuleName := ADR('Waterheater Energy'),
		Mode := mpENERGY_REG_MODE_COLLECT,
		Units := mpENERGY_ENERGY_UNIT_WS,
		ForwardActiveEnergy := ForwardActiveEnergy);

END_ACTION
```

#### AuditTrail.st - Watch water temperature for value change
```iecst
ACTION AuditTrail:

	// Manage recipe datapoints
	IF (WaterTemp <> _WaterTemp) THEN
		MpAuditValueChangeStatus := MpAuditValueChange(gAuditTrail, _WaterTemp, WaterTemp, '104');
		_WaterTemp := WaterTemp;
	END_IF

END_ACTION
```

### Program Logical/ConveyorSim (IEC) - Conveyor simulation

#### Cyclic.st - Cyclic code
```iecst
PROGRAM _CYCLIC
//	Cupfeed conveyor simulation
	IF (gCoffeeMainLogic.AxisCupFeeder.Active = TRUE)   THEN
		IF (gCoffeeMainLogic.AxisCupFeeder.Power = TRUE) THEN
			gCoffeeMainLogic.AxisCupFeeder.PowerOn 	:= TRUE;
			ActivePowerCupFeeder := 30;
			IF (gCoffeeMainLogic.AxisCupFeeder.MoveAdditive = TRUE) THEN
				IF (gCoffeeMainLogic.AxisCupFeeder.Position < 700.0) THEN
					gCoffeeMainLogic.AxisCupFeeder.Position 	:=
					gCoffeeMainLogic.AxisCupFeeder.Position + 1.5;
					ActivePowerCupFeeder := 80;
				ELSE
					gCoffeeMainLogic.AxisCupFeeder.InPosition := TRUE;

					ActivePowerCupFeeder := 30;
				END_IF;
			END_IF;
			Energy;
		ELSE
			gCoffeeMainLogic.AxisCupFeeder.PowerOn 	:= FALSE;
			ActivePowerCupFeeder := 0;
			Energy;
		END_IF;
	ELSE
		gCoffeeMainLogic.AxisCupFeeder.PowerOn 	:= FALSE;

		ActivePowerCupFeeder := 0;
		Energy;
	END_IF;

	//	Takeout conveyor simulation
	IF (gCoffeeMainLogic.AxisTakeout.Active = TRUE)   THEN
		IF (gCoffeeMainLogic.AxisTakeout.Power = TRUE) THEN
			gCoffeeMainLogic.AxisTakeout.PowerOn 	:= TRUE;
			ActivePowerTakeout := 10;
			IF (gCoffeeMainLogic.AxisTakeout.MoveAdditive = TRUE) THEN
				IF (gCoffeeMainLogic.AxisTakeout.Position < 300.0) THEN
					gCoffeeMainLogic.AxisTakeout.Position 	:=
					gCoffeeMainLogic.AxisTakeout.Position + 1.5;
					ActivePowerTakeout := 68;
				ELSE
					gCoffeeMainLogic.AxisTakeout.InPosition := TRUE;

					ActivePowerTakeout := 10;
				END_IF;
			END_IF;
			Energy;
		ELSE
			gCoffeeMainLogic.AxisTakeout.PowerOn 	:= FALSE;
			ActivePowerTakeout := 0;
			Energy;
		END_IF;
	ELSE
		gCoffeeMainLogic.AxisTakeout.PowerOn 	:= FALSE;

		ActivePowerTakeout := 0;
		Energy;
	END_IF;

END_PROGRAM
```

#### Init.st - Init code
```iecst
PROGRAM _INIT
	gCoffeeMainLogic.AxisTakeout.Active 	:= TRUE;
	gCoffeeMainLogic.AxisCupFeeder.Active 	:= TRUE;
END_PROGRAM
```

#### Energy.st - Record energy usage for water heater
```iecst
ACTION Energy:

	MpEnergyRegPower_0(
		MpLink := ADR(gEnergyCore),
		Enable := TRUE,
		ModuleName := ADR('ConveyorCupFeeder'),
		Mode := mpENERGY_REG_MODE_COLLECT,
		Units := mpENERGY_POWER_UNIT_W,
		ActivePower := ActivePowerCupFeeder);

	MpEnergyRegPower_1(
		MpLink := ADR(gEnergyCore),
		Enable := TRUE,
		ModuleName := ADR('ConveyorTakeout'),
		Mode := mpENERGY_REG_MODE_COLLECT,
		Units := mpENERGY_POWER_UNIT_W,
		ActivePower := ActivePowerTakeout);

END_ACTION
```

#### Variables.var
```iecst
VAR
	ActivePowerCupFeeder : INT := 0;
	MpEnergyRegPower_1 : MpEnergyRegPower := (0);
	ActivePowerTakeout : INT := 0;
	MpEnergyRegPower_0 : MpEnergyRegPower := (0);
END_VAR
```

- Visualisation Logical/mappView (not shown)

### Package Logical/UserFiles - Copy UserFiles to C:\mappDemo

### Coffee.st
```iecst
//MpCodeBox Program File (http:://www.br-automation.com)
//$Name:Coffee
//$Version:1.00.0
//$CodeType:MpLD
//$Created:2018-04-20 10:34,Anonymous
//$Changed:2018-04-20 10:34,Anonymous
//$Comment:
PROGRAM _INIT
END_PROGRAM
PROGRAM _CYCLIC
NETWORK 1 (* Add your comment here... *)
0[]:CONTACT:NO:StartPos()
1[0]:COIL:D:LampRed()
END_NETWORK
NETWORK 2 (* Add your comment here... *)
0[]:CONTACT:NO:EndPos()
1[0]:COIL:D:LampGreen()
END_NETWORK
END_PROGRAM
//$Sign:-
```

### Program Logical/Frequenza (IEC)

#### Cyclic.ld - Cyclic code
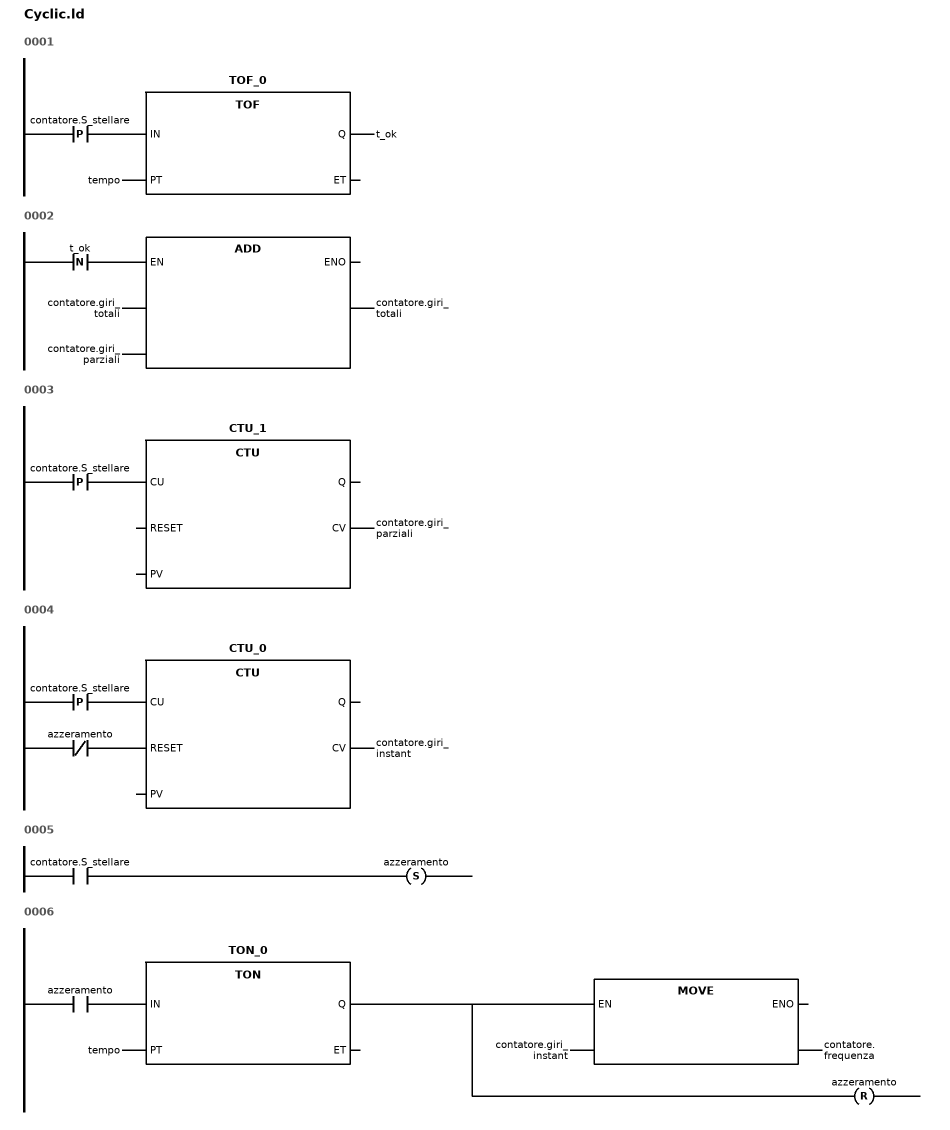
Ladder, written as Structured Text:
```iecst
PROGRAM _CYCLIC
VAR
    _e1 : R_TRIG;
    _e2 : F_TRIG;
    _e3 : R_TRIG;
    _e4 : R_TRIG;
END_VAR
(* Network 1 *)
_e1(CLK := contatore.S_stellare);
TOF_0(IN := _e1.Q, PT := tempo);
t_ok := TOF_0.Q;

(* Network 2 *)
_e2(CLK := t_ok);
IF _e2.Q THEN contatore.giri_totali := contatore.giri_totali + contatore.giri_parziali; END_IF;

(* Network 3 *)
_e3(CLK := contatore.S_stellare);
CTU_1(CU := _e3.Q);
contatore.giri_parziali := CTU_1.CV;

(* Network 4 *)
_e4(CLK := contatore.S_stellare);
CTU_0(CU := _e4.Q, RESET := NOT azzeramento);
contatore.giri_instant := CTU_0.CV;

(* Network 5 *)
IF contatore.S_stellare THEN azzeramento := TRUE; END_IF;

(* Network 6 *)
TON_0(IN := azzeramento, PT := tempo);
IF TON_0.Q THEN
    contatore.frequenza := contatore.giri_instant;
    azzeramento := FALSE;
END_IF;
END_PROGRAM
```

#### Variables.var - Local variables
```iecst
VAR
	CTU_0 : CTU := (0);
	TOF_0 : TOF := (0);
	tempo : TIME := T#1S;
	TON_0 : TON := (0);
	azzeramento : BOOL := FALSE;
END_VAR
```

### Program Logical/Conteggio (IEC)

#### Cyclic.st - Cyclic code
```iecst
PROGRAM _CYCLIC
	(* Insert code here *)

	DtSetTime_1.enable:=setta_orario;
	DtSetTime_1();
	//status:=DTGetTime_1.status;
	DtSetTime_1.DT1 := DT_attuale;

	DtGetTime_1.enable:=TRUE;
	DtGetTime_1();
	//status:=DTGetTime_1.status;
	DT_0:=DtGetTime_1.DT1;

	IF sim THEN

		IF conteggio THEN
			conteggio :=0;
			contatore.S_stellare:=0;
		ELSIF conteggio = 0 THEN
			conteggio := 1;
			contatore.S_stellare:=1;
		END_IF;
	ELSE

		contatore.S_stellare := contatore.Inp_S_Stellare;

	END_IF

	IF NOT t_ok THEN
		IF bool_1 = 1 THEN
			bool_1:=0;
			DT_2 := DT_0;
			tempo_attuale:=DiffDT(DT_2,DT_1);
			StartGenerate := 1;
		END_IF;
	ELSE
		IF bool_1 = 0 THEN
			DT_1 := DT_0;
		END_IF;

		bool_1 := 1;
	END_IF;

	IF MpReportCore_0.CommandDone THEN CTU_1.RESET := 1; ELSE CTU_1.RESET := 0; END_IF;

	Ricetta.Giri_Parziali	:= contatore.giri_parziali;
	Ricetta.Giri_Totali		:= contatore.giri_totali;
	Ricetta.Ora_Fine		:= DT_2;
	Ricetta.Ora_Inizio		:= DT_1;
	Ricetta.Tempo_Attivita	:= tempo_attuale;

	contatore.nome_ricetta	:= DT_TO_STRING(DT_1);
//	contatore.nome_ricetta2 := contatore.nome_ricetta;

END_PROGRAM
```

#### Variables.var - Local variables
```iecst
VAR
	DtSetTime_1 : DTSetTime := (0);
	DtGetTime_1 : DTGetTime := (0);
	DT_2 : DATE_AND_TIME := DT#1970-01-01-00:00:00;
	DT_0 : DATE_AND_TIME := DT#1970-01-01-00:00:00;
	DT_attuale : DATE_AND_TIME := DT#1970-01-01-00:00:00;
	DT_1 : DATE_AND_TIME := DT#1970-01-01-00:00:00;
	tempo_attuale : UDINT := 0;
	totale : UDINT := 0;
	parziale : UDINT := 0;
	bool_1 : BOOL := FALSE;
	sim : BOOL := FALSE;
	setta_orario : BOOL := FALSE;
	conteggio : BOOL := FALSE;
END_VAR
```

### Program Logical/Program (ANSIC)

#### Cyclic.c - Cyclic code
```c
#include <bur/plctypes.h>

#ifdef _DEFAULT_INCLUDES
	#include <AsDefault.h>
#endif

void _CYCLIC ProgramCyclic(void)
{
	contatore.nome_ricetta3 = memcpy((&contatore.nome_ricetta2),(&contatore.nome_ricetta),sizeof(contatore.nome_ricetta));

	contatore.nome_ricetta2[0] 		= 'R';
	contatore.nome_ricetta2[1] 		= 'P';
	contatore.nome_ricetta2[16] 	= '_';
	contatore.nome_ricetta2[19] 	= '_';
}
```

Listed in the project but not available here: Logical/Infrastructure/Report/Types.typ, Logical/Infrastructure/IO/Types.typ, Logical/Frequenza/Init.ld, Logical/Frequenza/Exit.ld, Logical/Frequenza/Types.typ, Logical/Conteggio/Init.st, Logical/Conteggio/Exit.st, Logical/Conteggio/Types.typ, Logical/Program/Init.c, Logical/Program/Exit.c, Logical/Program/Types.typ, Logical/Program/Variables.var
